// debug log
LogLvl(Lvl:=E_LogSeverity.Debug, F_Concat4('printStart: at XS:', TO_STRING(_nPosXS), ' ', _pNewAttached^.print(0)));  // print container
LogLvl(Lvl:=E_LogSeverity.Debug, F_Concat4(
                                      F_Concat3('> XS = X0(', TO_STRING(iCT.GetPosX0(iTracker:=_iCTTracker)), ')'),
                                      '',
                                      F_Concat3(' + shStartOffs(', TO_STRING(F_MeterToSubPixel(fPrintStartOffset, _fPrintResolution*_fSubPxResolution)), ')'),
                                      F_Concat3(' - shDropComp(', TO_STRING(F_MeterToSubPixel(fbDropSpeedComp.fDropPlacementError, _fPrintResolution*_fSubPxResolution)), ')')
                                   ));

// debug history
FOR i:=0 TO nC_HistorySize-1 DO sRepeatHistory[i].bSelected := FALSE; END_FOR   // clear selection
nRepeatCt := (nRepeatCt + 1) MOD nC_HistorySize;
sRepeatHistory[nRepeatCt].bSelected      := TRUE;
sRepeatHistory[nRepeatCt].nX0            := _nPosXS;
sRepeatHistory[nRepeatCt].fLen           := _pNewAttached^.pJob^.fImageDepth;  // + PrePost?
sRepeatHistory[nRepeatCt].fLenEffective  := _nPosXS - sRepeatHistory[SEL(nRepeatCt=0, nRepeatCt-1, nC_HistorySize-1)].nX0;
END_METHOD

PROPERTY bGridWasLimited : BOOL
GET
bGridWasLimited := _bGridWasLimited;
END_GET
END_PROPERTY

PROPERTY bJobActive : BOOL
GET
bJobActive := _bJobActive;
END_GET
END_PROPERTY

PROPERTY bPausePrintCanEx : BOOL
GET
bPausePrintCanEx := FALSE; //Not implemented
END_GET
END_PROPERTY

PROPERTY bPcEnabled : BOOL
GET
bPcEnabled := fB_PcAdapter.bPcEnable;
END_GET
END_PROPERTY

PROPERTY bPrintEnabled : BOOL
GET
bPrintEnabled := _bEnable;
END_GET
END_PROPERTY

PROPERTY bPrinting : BOOL
GET
bPrinting := fbPa.bPrinting;
END_GET
END_PROPERTY

PROPERTY bPrintReady : BOOL
GET
bPrintReady := fbPa.bReady;
END_GET
END_PROPERTY

PROPERTY bQueueEmpty : BOOL
GET
bQueueEmpty := NOT fB_PcAdapter.bJobValid;
END_GET
END_PROPERTY

PROPERTY bStartPrintCanEx : BOOL
GET
bStartPrintCanEx := fbPa.bStartCanEx;
END_GET
END_PROPERTY

PROPERTY bStopPrintCanEx : BOOL
GET
bStopPrintCanEx := fbPa.bStopCanEx;
END_GET
END_PROPERTY

{attribute 'monitoring':='call'}
PROPERTY bWorkerEnable : BOOL
GET
bWorkerEnable := SUPER^.bWorkerEnable;
END_GET
SET
IF _pAdsPg = 0 THEN
  SUPER^.bWorkerEnable := bWorkerEnable;
ELSE
  // mask worker enable with group enable
  SUPER^.bWorkerEnable := bWorkerEnable AND _pAdsPg^.bEnable;  
END_IF
END_SET
END_PROPERTY

{attribute 'monitoring':='call'}
PROPERTY bWorkerPrintEnable : BOOL
GET
bWorkerPrintEnable := _bWorkerPrintEnable;
END_GET
SET
_bWorkerPrintEnable := bWorkerPrintEnable;
END_SET
END_PROPERTY

(*
  Check timing for grid stream. 
  Reports an error if grid stream is too slow (machine running too fast for streaming the grid points over PDI)
  :returns: TRUE on error
*)
METHOD PRIVATE checkGridTiming : BOOL
VAR_INPUT
  nPosXS : DINT;
  nPosNow : DINT;
END_VAR
// check for timing problems
IF fMasterSpeed <> 0 THEN

  // - check pre-charge at beginning
  IF _fColumnsToPrecharge * fC_GRIDPOINT_STREAM_TIME * _sPhGridHwCfg.nGridRoiRows >= F_SubPixelToMeter(lPosSubPx:=SEL(nPosXS-nPosNow>0, 0, nPosXS-nPosNow), fResSubPx:=_fPrintResolution*_fSubPxResolution) / fMasterSpeed  THEN
    checkGridTiming := TRUE;
    LogError('Machine too fast for grid stream (for pre-charge at attach)');
  END_IF
  
  // - check charge time needed per columns vs machine speed and grid-sizeY
  IF fC_GRIDPOINT_STREAM_TIME * _sPhGridHwCfg.nGridRoiRows >= F_SubPixelToMeter(lPosSubPx:=TO_DINT(sDefGridSettings.nGridPitchX), fResSubPx:=_fPrintResolution) / fMasterSpeed THEN
    checkGridTiming := TRUE;
    LogError('Machine too fast for grid stream (time rows per column)');
  END_IF

END_IF
END_METHOD

(*
  Check if intended print position is valid. 
  - Reports an error if print start position is not in the future
  :returns: TRUE on error
*)
METHOD checkPrintposTiming : BOOL
VAR_INPUT
  nStartPos   : DINT;   // intended start position
  nCurrentPos : DINT;   // current position
END_VAR
IF (nStartPos - nCurrentPos) < 0 THEN 
  checkPrintposTiming := TRUE;
  LogWarning(Msg:=F_Concat4('Print start position:', TO_STRING(nStartPos) ,' < Encoder position:', TO_STRING(nCurrentPos)));
END_IF
END_METHOD

// apply other corrections to camera correction/deformation
METHOD PRIVATE correctionApply : BOOL
VAR_INPUT
  pPoint : POINTER TO ST_DeformationPointAccurate;
END_VAR
VAR
  i : UDINT;
END_VAR

// here apply all PU specific corrections
// - mechanical stretch based on temperature extension (if not done in Camera)
// - banana correction
// - Y-shifts of PU
// - trapzedoial correction
// - ...


// PU Deformation correction
IF GVL_Deformation.bC_UsePUDeformation THEN
  FOR i:=1 TO nPointCorrections DO
    iPointCorrections[i].updateCorrection(pPoint:=pPoint);
  END_FOR
END_IF
END_METHOD

(*
  Limit correction to boundaries
  :return: TRUE if limited
*)
METHOD PRIVATE correctionLimit : BOOL
VAR_INPUT
  pPoint : POINTER TO ST_DeformationPointAccurate;
  pCT    : POINTER TO FB_ContainerDefGrid;
END_VAR
VAR
  bLimited : BOOL;
  nExeedX, nExeedY : LREAL;
END_VAR
// limit point correction to boundaries and inform
IF pPoint^.dx >= _fLimitCorrectionX    THEN nExeedX := pPoint^.dx; pPoint^.dx := _fLimitCorrectionX;    bLimited:=TRUE; END_IF
IF pPoint^.dx <= -1*_fLimitCorrectionX THEN nExeedX := pPoint^.dx; pPoint^.dx := -1*_fLimitCorrectionX; bLimited:=TRUE; END_IF
IF pPoint^.dy >= _fLimitCorrectionY    THEN nExeedY := pPoint^.dy; pPoint^.dy := _fLimitCorrectionY;    bLimited:=TRUE; END_IF
IF pPoint^.dy <= -1*_fLimitCorrectionY THEN nExeedY := pPoint^.dy; pPoint^.dy := -1*_fLimitCorrectionY; bLimited:=TRUE; END_IF

IF bLimited THEN
  LogLvl(Lvl:=E_LogSeverity.Debug, Msg:=F_Concat4( F_concat2('Correction limited - Point=',TO_STRING(pPoint^.index)),
                                                     F_Concat5(' (c:',TO_STRING(pPoint^.col),'/r:',TO_STRING(pPoint^.row), ') '),
                                                     F_Concat4('dx:', TO_STRING(nExeedX), 'px dy:', TO_STRING(nExeedY)),
                                                     F_Concat4('px dx_max=+/-', TO_STRING(_fLimitCorrectionX), ' dy_max=+/-', TO_STRING(_fLimitCorrectionY))
                                                  ));
END_IF

_bGridWasLimited := SEL(bLimited, FALSE, TRUE);
correctionLimit := bLimited;
END_METHOD

// current job image length in [m]
PROPERTY fImageLength : LREAL
GET
fImageLength := _fCurrentImgDepth;
END_GET
END_PROPERTY

PROPERTY fMaxPrintSpeed : LREAL
GET
fMaxPrintSpeed := 0;  // TODO: when i_pc_adapter has the info from pc/ph
END_GET
END_PROPERTY

(*
  Max. supported speed [m/s], 0 if not available
*)
{attribute 'monitoring':='call'}
PROPERTY fMaxSpeed : LREAL
GET
VAR
  nSpeedMpMin : DINT;
END_VAR
nSpeedMpMin := SEL(bWorkerEnable AND _pAdsPg <> 0, 0, _pAdsPg^.lMaxPrintSpeed);
fMaxSpeed := TO_LREAL(nSpeedMpMin)/60;
END_GET
END_PROPERTY

{attribute 'monitoring':='call'}
PROPERTY fStartShiftFactor : LREAL
GET
fStartShiftFactor := _fStartShiftFactor;
END_GET
SET
_fStartShiftFactor := fStartShiftFactor;
END_SET
END_PROPERTY

{attribute 'monitoring':='call'}
PROPERTY fStartShiftOffset : LREAL
GET
fStartShiftOffset := _fStartShiftOffset;
END_GET
SET
_fStartShiftOffset := fStartShiftOffset;
END_SET
END_PROPERTY

METHOD PROTECTED gridUpdate : BOOL
VAR_INPUT
  bEnableDeformation : BOOL;      // enable correction update, else correction (0/0) is written
  pCT : POINTER TO FB_ContainerDefGrid;
  pCTHdlData : POINTER TO ST_WorkerDefGrid_CTData;
  pMaxDx : POINTER TO LREAL;
END_VAR
VAR
  bOK : BOOL;
  fCurrentColumnPos  : LREAL; // Currently column position (of current ct)
END_VAR


//TODO: rewrite this method to look cleaner (less if else)
IF sDefGridSettings.nGridSizeX  = 0 THEN RETURN; END_IF          // avoid endless loops
IF sDefGridSettings.nGridSizeY  = 0 THEN RETURN; END_IF
IF sDefGridSettings.nGridPitchX = 0 THEN RETURN; END_IF
IF pCT = 0 THEN RETURN; END_IF
IF pCTHdlData = 0 THEN RETURN; END_IF

gridUpdate:=TRUE;

// calculate grid column position
fCurrentColumnPos := pCTHdlData^.fPosRelToAttach / (sDefGridSettings.nGridPitchX * _fSubPxResolution);   // calc grid column position relative to worker

// Check for next correction update
bOK := TRUE;
IF pCTHdlData^.nChargedCols <= sDefGridSettings.nGridSizeX THEN
  IF bEnableDeformation THEN 
    // sync deformation points
    bOK := streamCorrection(pCT:=pCT,
                            fColPos := fCurrentColumnPos, 
                            pChargedCols:=ADR(pCTHdlData^.nChargedCols), 
                            pMaxDx:=pMaxDx,
                            nAvailPoints:=pCT^.nAvailableGridPoints);
  ELSE
    // sync empty deformation points (with NO correction)
    bOK := streamNoCorrection(pChargedCols:=ADR(pCTHdlData^.nChargedCols));
  END_IF
  
END_IF

gridUpdate := bOK;
END_METHOD

METHOD InitWorkerPrint : BOOL
VAR_INPUT
  pAdsPg                : POINTER TO FB_ADS_PG;       // pg ads reference (worker prints ads)
  iDefGridParamMediator : I_ParamMediator;            // for deformation settings
  fLimitCorrectionX     : LREAL;                      // correction limit in y (abs) [px]
  fLimitCorrectionY     : LREAL;                      // correction limit in y (abs) [px]
END_VAR
IF NOT bInitialized            THEN LogError('Base Worker not initialized! call init() before'); RETURN; END_IF
IF pAdspg = 0 THEN LogError('InitWorkerPrint: invalid parameter proviced'); RETURN; END_IF
IF iDefGridParamMediator = 0   THEN bInitialized := FALSE; LogError('Invalid parameter, no valid param mediator'); RETURN; END_IF

// Worker specific init
_pAdsPg := pAdsPg;
_iParamMediator := iDefGridParamMediator;

_fLimitCorrectionX := ABS(fLimitCorrectionX);
_fLimitCorrectionY := ABS(fLimitCorrectionY);

// Print Aggregate
fbPa.bSyncAfterDone := FALSE;
fbPa.init(iPcAdapter := fB_PcAdapter, iPsInterface := fbPs);
END_METHOD

METHOD mJobPause
END_METHOD

METHOD   mJobStart
VAR_INPUT
	sJobDef	: CalmarCompPrint.I_JobDefinition;
END_VAR
// Config workers static variables
// - security release position (2 * Image Length)
_fCtSecurityReleasePos := F_MeterToSubPixel(fPosMeter:=2.1*(sJobDef.fImageDepth/1000), fResoSubPx:=_fPrintResolution*_fSubPxResolution);

IF NOT bWorkerEnable THEN RETURN; END_IF  // only if enabled

// an initial definition at jobStart/(activation)
fbPs.setupObject(nObjId:=1, nCopy:=1, bStop:=FALSE, bDir:=FALSE, nPrintStartPos:=0, nImageSelection:=0, nShiftedStartX:=0);
fbPa.jobStart(bEndless:=sJobDef.isEndless());

_fCurrentImgDepth := sJobDef.fImageDepth/1000;
_bEndless := sJobDef.isEndless();
bBuffStopBit := NOT _bEndless;

// update deformation limit by job setting
//_fLimitCorrectionX   // [px]

// grid settings update
IF _iPhGrid <> 0 THEN _sPhGridHwCfg := _iPhGrid.getGridHwCfg(); END_IF 

_bJobActive := TRUE;
END_METHOD

METHOD  mJobStop
VAR_INPUT
	sStatus	: CalmarCompPrint.I_JobStatus;
END_VAR
fbPa.jobStop();
_bJobActive := FALSE;
_bPaStarted := FALSE;
_bPaStartRequested := FALSE;
END_METHOD

METHOD mProduced
VAR_INPUT
	(* current progress*)
	sProgress	: CalmarCompPrint.I_JobProgress;
END_VAR
END_METHOD

// register additional grid correction handlers
METHOD RegisterGridCorrection : BOOL
VAR_INPUT
  iGridCorrection : I_GridPointCorrection;
END_VAR
VAR
  i : UDINT;
END_VAR
IF iGridCorrection = 0 THEN LogError('registerGridCorrection: ivalid interface, ignore'); RETURN; END_IF
IF nPointCorrections >= nC_NUM_POINTCORRECTIONS THEN LogError('registerGridCorrection: too many corrections registred, ignore'); RETURN; END_IF

nPointCorrections := nPointCorrections + 1;
iPointCorrections[nPointCorrections] := iGridCorrection;
END_METHOD

METHOD registerPc : BOOL
VAR_INPUT
  iNewPC : I_PC;
END_VAR
registerPc := fB_PcAdapter.registerPc(iNewPC := iNewPC);
END_METHOD

METHOD registerPh : BOOL
VAR_INPUT
  iPH : I_PH;
END_VAR
//Attach head to print station
IF iPH <> 0 THEN
  fbPs.registerPh(iNewPh:=iPH);
  _iPhGrid := iPH.iGridCorrection;
END_IF
END_METHOD

(*
  Release CT from Worker.
  :return: TRUE if CT was released, FALSE if no CT was registered 
*)
METHOD Release : BOOL
VAR_INPUT
  iCT              : I_CT;                         (*container at triggered event position*)
END_VAR

Release := SUPER^.Release(iCT:=iCT);
END_METHOD

// Release all attached CTs
METHOD PRIVATE ReleaseAllAttached
VAR
  i : UDINT;
  pCt : POINTER TO FB_ContainerDefGrid;
END_VAR
//Work only with attached container
IF _nAttachedCTs = 0 THEN RETURN; END_IF
  
FOR i:=nLowerIndexCTList TO nLowerIndexCTList + _nAttachedCTs - 1 DO
  pCt := _pAttachedCTList[i];
  pCt^.AbortDeformation(sReason:=EC_Print.ecPaAbortHold.Desc, Src:=_pEcSrc^, bHideLog:=TRUE);
  
  Release(iCT:=pCt^);
END_FOR
END_METHOD

METHOD PRIVATE setupPosition
VAR
  fPreStartShift : LREAL;
  fCalculatedWorkerPos : LREAL;
END_VAR
IF _pAttachedCt <> 0 THEN RETURN; END_IF   // Update only without attached container

// Worker position update
fPreStartShift := (_fStartShiftOffset + _fStartShiftFactor * fMasterSpeed);
fCalculatedWorkerPos := fPrintStartOffset + fPreStartShift;
IF _fWorkerPosition <> fCalculatedWorkerPos THEN   // Worker position changed
  fPosition := fCalculatedWorkerPos;  // Update worker position
END_IF
END_METHOD

METHOD PRIVATE sim
END_METHOD

METHOD PRIVATE streamCorrection : BOOL
VAR_INPUT
  pCT : POINTER TO FB_ContainerDefGrid;
  fColPos : LREAL;  // current column position (relative to Attach-Pos)
  pChargedCols : POINTER TO UDINT;  // number of already charged columns (pointer for internal edit)
  pMaxDx : POINTER TO LREAL;
  nAvailPoints : UDINT;     // available gridPoints on CT
END_VAR
VAR
  nRow : UDINT;
  bWasSet : BOOL;
  sPoint : ST_DeformationPointAccurate;
  fCurrentPreCharge  : LREAL; // Currently to be precharged (for scope)
END_VAR
VAR_INST
  nAvailPoints_mem : UDINT;
END_VAR
IF pChargedCols = 0 THEN RETURN; END_IF

streamCorrection := TRUE;

fCurrentPreCharge := fColPos + _fColumnsToPrecharge;

WHILE pChargedCols^ < LIMIT(0, FLOOR(fCurrentPreCharge), sDefGridSettings.nGridSizeX) DO
  
  IF nAvailPoints >= sDefGridSettings.nGridSizeY * (pChargedCols^+1) THEN     // Complete next column available?
    
    nAvailPoints_mem := 0;
    LogLvl(Lvl:=E_LogSeverity.Debug, Msg:=F_Concat4('CT: ', TO_STRING(pCT^.pCT^.iId),' Charge CG col: ', TO_STRING(pChargedCols^)));
    
    pMaxDx^ := 0;   // per columns
    
    FOR nRow := 0 TO sDefGridSettings.nGridSizeY - 1 DO
      
      // get points
      IF pCT^.getDeformationPoint(nCol:=pChargedCols^, nRow:=nRow, nSel:=0, sPoint=>sPoint, bWasSet=>bWasSet) THEN
        
        IF NOT bWasSet THEN LogWarning(F_Concat5('Point[c(',TO_STRING(pChargedCols^),')/r(', TO_STRING(nRow),')] was not set')); END_IF
        
        // apply PU corrections
        correctionApply(pPoint:=ADR(sPoint));
        
        // limitation corrections
        correctionLimit(pPoint:=ADR(sPoint), pCT:=pCt);
        
        // max. dx tracing
        IF sPoint.dx > pMaxDx^ THEN pMaxDx^ := sPoint.dx; END_IF
        
        // send point
        IF NOT fbPs.newGridPoint(sPoint:=sPoint) THEN
          // err
          LogError(Msg:='stream new point failed');
          streamCorrection:=FALSE;
          RETURN;
        ELSE
          // ok
          pCT^.storeStreamedDeformationPoint(pPoint:=ADR(sPoint));    // save to sent table
          IF bEnVerbose THEN
            F_Concat3( 
              F_concat2('Send Point=',TO_STRING(sPoint.index)),
              F_Concat5(' (c:',TO_STRING(sPoint.col),'/r:',TO_STRING(sPoint.row), ')'),
              F_Concat4(' dx=', TO_STRING(sPoint.dx), ' dy=', TO_STRING(sPoint.dy))
            );
          END_IF
        END_IF
      ELSE
        LogError(Msg:='get new grid point failed');
        streamCorrection:=FALSE;
      END_IF
    END_FOR
    
    pChargedCols^ := pChargedCols^ + 1;
  ELSE
    
    // not yet enought points for next full column
    IF nAvailPoints > nAvailPoints_mem THEN // log once or after every update of new available points
      LogLvl(Lvl:=E_LogSeverity.Error, Msg:=F_Concat3(
                                            F_Concat2('CT: ', TO_STRING(pCT^.pCT^.iId)), 
                                            F_Concat2(' Print column expected but not available. Avil=', TO_STRING(nAvailPoints)),
                                            F_Concat2(' of expected: ', TO_STRING(sDefGridSettings.nGridSizeY * (pChargedCols^+1)))
                                          ));
    END_IF
    nAvailPoints_mem := nAvailPoints;
    streamCorrection:=FALSE;
    RETURN;
  END_IF
  
END_WHILE
END_METHOD

METHOD PRIVATE streamNoCorrection : BOOL
VAR_INPUT
  pChargedCols : POINTER TO UDINT;  // number of already charged columns (pointer for internal edit)
END_VAR
VAR
  nRow : UDINT;
  sPoint : ST_DeformationPointAccurate;
END_VAR
IF pChargedCols = 0 THEN RETURN; END_IF

// send points with no deformation
FOR nRow := 0 TO sDefGridSettings.nGridSizeY - 1 DO
    MEMSET(destAddr:=ADR(sPoint), fillByte:=0, n:=SIZEOF(sPoint));
    sPoint.col := TO_DINT(pChargedCols^);
    sPoint.row := TO_DINT(nRow);
    IF NOT fbPs.newGridPoint(sPoint:=sPoint) THEN
       LogError(Msg:='stream new point failed');
       streamNoCorrection:=FALSE;
       RETURN;
    END_IF
END_FOR

// select next column
pChargedCols^ := pChargedCols^ + 1;

streamNoCorrection := TRUE;
END_METHOD

METHOD work
VAR
  bDeformErr : BOOL;
  nDeformStep : E_DeformationStep;
  i : UDINT;
  pCt : POINTER TO FB_ContainerDefGrid;
  pCtHdlData : POINTER TO ST_WorkerDefGrid_CTData;
  nUpdateStopPos : DINT;
  fMaxDx : LREAL;
END_VAR
IF _iParamMediator = 0 THEN F_Report_Error(ErrType:=EN_REPORT_ERROR_TYPE.Report_Error_0Pointer); RETURN; END_IF
bError := FALSE; nError := 0;

setupPosition();  // calculate and set worker position

SUPER^.work();

(*Print correction*)
fbDropSpeedComp(fMasterSpeed:=fMasterSpeed, fDropTravelDistance:=fPUElevation);

(*Update virtual encoder on all controller boards*)
fB_PcAdapter.setEncoderPos(nPrintPos);
fB_PcAdapter();

(*Call print aggregate*)
rTrigHwSync(CLK:=bHardwareSync); 
IF rTrigHwSync.Q THEN fbPa.sync(); END_IF   // external sync cmd

// PA control
fbPa.bHold := bHardwareHold;                // external hw hold, NOTE: this stop the current print iPC.stop()
fbPa();
PaStartTimeout(IN:=_bPaStartRequested, PT:=fbPa.fbStatePrepare.tC_PrepareTimeout+T#10MS);

IF _bPaStartRequested THEN
  // Starting...
  IF fbPa.bPrinting THEN
    // started
    _bPaStarted := TRUE; 
    _bPaStartRequested := FALSE;
  ELSIF PaStartTimeout.Q THEN     // Abort print
    // start timeout -> abort
    _bPaStarted := FALSE;
    _bPaStartRequested := FALSE;
    fbPa.printStop(bSyncedStop:=FALSE);
    ReleaseAllAttached();
  END_IF
ELSIF _bPaStarted THEN
  // - Started... Supervision of FSM
  IF fbPa.bDone OR fbPa.bStop THEN  // if pa did stop
    _bPaStarted := FALSE; 
    ReleaseAllAttached();
  (*ELSIF fbpa.bError THEN
    ReleaseAllAttached();*)
	END_IF 
  // - disabled
  IF NOT bWorkerEnable THEN
    _bPaStarted := FALSE;
    fbPa.printStop(bSyncedStop:=FALSE);
    ReleaseAllAttached();
  END_IF
  // - machine stopped
  IF bFastStopRequest OR bHardwareHold THEN
    _bPaStarted := FALSE;
    fbPa.printStop(bSyncedStop:=FALSE);
    ReleaseAllAttached();
	END_IF
  // - Synced stopping request
  IF bPrintStopRequest THEN
    IF NOT _bPaStopping THEN  _bPaStopping := TRUE;
      fbPs.stopObject(nObjId:=0, 
                      nStopPosition:=   _nPosXS           // use last used/calculated XS
                                      + F_MeterToSubPixel(fPosMeter:=_fCurrentImgDepth + 0.05, fResoSubPx:=_fPrintResolution*_fSubPxResolution)
                                      + TO_DINT(nPhDepth*_fSubPxResolution));
      fbPa.printStop(bSyncedStop:=TRUE);                  // should stop automatically when all buffer are done   
     END_IF
  ELSE
    _bPaStopping := FALSE;
  END_IF
END_IF

bPrintActive := _bPaStarted;


// for all attached CTs ----------------
// - Disable      -> PA.Stop, tag all as error, release all [OK]
// - FastStop     -> PA.Stop, tag all as error, release all [  ]
// - Hold         -> PA.Hold => PC.stop() [  ]
// - PA Starting  ->  [  ]
// - JobStop      -> PA.jobStop() -> tag all as error, release all [  ]
// - Normal Stop  -> PS.Request a stop [  ]
// - OK           =>  GridStream -> Release when all done [  ]
FOR i:=nLowerIndexCTList TO nLowerIndexCTList + _nAttachedCTs - 1 DO
  pCt := _pAttachedCTList[i];
  // Handling Data
  // - fPosRelToAttach: position relative to attach
  // - nChargedCols: charged columns
  // - nData2: not used
  // - fData1: not used
  // - fData2: not used
  pCtHdlData := ADR(_stAttachedCTData[i]);
  
  // Grid update
  bDeformErr := pCt^.getDeformationStatus(eDStep=>nDeformStep);
  IF NOT bDeformErr AND nDeformStep >= E_DeformationStep.gridStarted AND NOT _bForceDefGridOff THEN
    IF NOT gridUpdate(bEnableDeformation:=TRUE, pCT:=pCt, pCTHdlData:=pCtHdlData, pMaxDx:=ADR(fMaxDx)) THEN
      pCt^.AbortDeformation(sReason:='deformation point update failed', Src:=_pEcSrc^, bHideLog:=FALSE);
    END_IF
  ELSE
    // not started or error already --> erase deformation points and send no correction points
    IF NOT gridUpdate(bEnableDeformation:=FALSE, pCT:=pCt, pCTHdlData:=pCtHdlData, pMaxDx:=ADR(fMaxDx)) THEN
      pCt^.AbortDeformation(sReason:='deformation point update failed', Src:=_pEcSrc^, bHideLog:=FALSE);
    END_IF
  END_IF
  
  // RELEASE when Grid stream finished
  IF pCtHdlData^.nChargedCols >= sDefGridSettings.nGridSizeX THEN
    IF NOT _bEndless THEN // single print mode
      // Update print length in single print mode
      nUpdateStopPos := pCtHdlData^.nXS                                                                                   // XS print start position
                      + F_MeterToSubPixel(fPosMeter:=_fCurrentImgDepth, fResoSubPx:=_fPrintResolution*_fSubPxResolution)  // sheet length
                      + F_MeterToSubPixel(fPosMeter:=fMaxDx, fResoSubPx:=_fPrintResolution)                               // max. deformation
                      + TO_DINT(nPhDepth*_fSubPxResolution);
      fbPs.stopObject(nObjId:=0, nStopPosition:=nUpdateStopPos);        // update (overwrite firmware internal calculated) jm stop position
      LogLvl(Lvl:=E_LogSeverity.Debug, Msg:=F_Concat6('Update StopPos=', TO_STRING(nUpdateStopPos),' (',F_UDINT_TO_HEXSTR(lVal:=TO_UDINT(nUpdateStopPos), bLower:=FALSE), ') on ', pCt^.print(format:=0)));
    END_IF
    Release(pCt^);
  END_IF
END_FOR


// forward pa state to pg ads
IF _pAdsPg <> 0 THEN
  _pAdsPg^.aState := fbPa.aPaState;
  _pAdsPg^.lError := nError; 
  _pAdsPg^.bError := bError;
END_IF


// logging config
fbPa.LogLevel := LogLevel;
fB_PcAdapter.LogLevel := LogLevel;

sim();
END_METHOD

END_FUNCTION_BLOCK

// ---- POUs/Print/WEU/FB_PrintModule_WEU_View.TcPOU
FUNCTION_BLOCK FB_PrintModule_WEU_View
VAR
  // helper
  bInit   : BOOL;
  
  // config
  _pModule : POINTER TO FB_PrintModule_WEU;
  _pPositioning : POINTER TO FB_PrintPositionDmax;
  
  fbCTTrackerView : FB_CTTrackerView;
  
  // view selections
  nSelWorkerPrint : UDINT := 1;
  bShowFineAlignement : BOOL;
  // hardware view
  bShowPhDetail : BOOL;
  nSelPhDetail : UDINT := 1;
  bShowPcDetail : BOOL;
  nSelPcDetail : UDINT := 1;
  
  // motion and position view
  bShowPositionDetail : BOOL;
  bMovingInd : BOOL;
  fSpeed  : LREAL;
  fbBlink_Moving : FB_BLINK;
  
  // debug view
  bShowDebugAndSim : BOOL;
  
  fbBlink_Printing : FB_BLINK;
  bBlinkPrint : BOOL;
  bPrintInd : ARRAY[1..GVL_WEU.nC_MaxWorkerPrintPerPm] OF BOOL;
  fMaxPos : LREAL;
  t : TIME;
  zPos_PM : UDINT;
  i : UDINT;
END_VAR

VAR CONSTANT
  nC_MAX_WORKER_VIEWS : UINT := 10;
END_VAR

IF NOT checkConfig() THEN RETURN; END_IF    // check config

// -- show moving -----------------------
fSpeed := _pPositioning^.getSpeed();
IF LrealIsNaN(x:=fSpeed) THEN
  fSpeed := 0;
END_IF
t := LREAL_TO_TIME(1000-fSpeed*900);
fbBlink_Moving(bI_Enable:=SEL(fSpeed > 0, FALSE, TRUE), tI_Time:=t, bO_Out=>bMovingInd);

t := T#400MS;
fbBlink_Moving(bI_Enable:=TRUE, tI_Time:=t, bO_Out=>bBlinkPrint);
FOR i:=1 TO GVL_WEU.nC_MaxWorkerPrintPerPm DO
  bPrintInd[i] := _pModule^.fbWorkerPrint[i].bPrinting AND bBlinkPrint;
  fMaxPos := MAX(_pModule^.fbWorkerPrint[i].fPosition, fMaxPos);
END_FOR


// -- show pm module position
zPos_PM := SEL(_pModule^._pModuleMachineState^.bUnitInPrintPosition, 0, 40);

// -- show pg in p,
nSelWorkerPrint := LIMIT(1, nSelWorkerPrint, GVL_WEU.nC_MaxWorkerPrintPerPm);

// -- show ph detail
nSelPhDetail := LIMIT(1, nSelPhDetail, _pModule^._nPh);
nSelPcDetail := LIMIT(1, nSelPcDetail, _pModule^._nPc);

// -- CTTracker overview view
fbCTTrackerView.fX_m  := fMaxPos + 0.1;
fbCTTrackerView.fY_m  := 1;
fbCTTrackerView.nX_px := 300;
fbCTTrackerView.nY_px := 100;
fbCTTrackerView.fPxToMRatio := fbCTTrackerView.nX_px / fbCTTrackerView.fX_m;
fbCTTrackerView.iPrintPosition :=_pPositioning^;
fbCTTrackerView();

METHOD checkConfig : BOOL
VAR_INPUT
END_VAR
VAR_INST
  _fX_m, _fY_m   : LREAL;
  _nX_px, _nY_px : DINT; 
END_VAR
VAR
  bOK : BOOL;
END_VAR
IF NOT bInit THEN RETURN; END_IF

checkConfig := TRUE;
END_METHOD

METHOD init : BOOL
VAR_INPUT
  pModule : POINTER TO FB_PrintModule_WEU;
  pPositioning : POINTER TO FB_PrintPositionDmax;
END_VAR
IF pPositioning = 0 OR pModule = 0 THEN RETURN; END_IF

_pModule := pModule;
_pPositioning := pPositioning;

// cttracker overview
fbCTTrackerView.init(pCTTracker:=ADR(_pModule^.fbCTTracker));

bInit := TRUE;
END_METHOD

END_FUNCTION_BLOCK

// ---- POUs/Print/obsolete/FB_DRIFTCONTROL.TcPOU
FUNCTION_BLOCK FB_DRIFTCONTROL
VAR_INPUT
  bI_Reset                    : BOOL;            (*reset fb and controller*)
  bI_Enable                   : BOOL;            (*[internal] auto enable of control*)
  bI_OutputEnable             : BOOL;            (*enable control output or 1.0 if off*)
  bI_RegisterMark             : BOOL;            (*start trigger (e.g. register mark)*)
  
  lI_RegisterMarkPosition     : DINT;            (*[Subpixel] Mark position*)
  lI_RefPosition              : DINT;            (*[Subpixel] Refereence position*)
  lI_ImgPosition              : DINT;            (*[Subpixel] Image position*)
(*UNUSED*)  fI_RefPosition            : LREAL;          (*[um] Refereence position*)    
(*UNUSED*)  fI_ImgPosition            : LREAL;          (*[um] Image position*)

  iI_Res_Ph                   : INT;             (*[dpi] resolution printhead native*)
  iI_Res_SubPix               : INT;             (*[-] resolution subpixel*)
  pI_JobSettings              : POINTER TO ST_JobSettings;
  
  fI_ControllerPGain          : LREAL := 0.5;    (*PDI controller P-Gain*)
  fI_ControllerIGain          : LREAL := 20;     (*PDI controller I-Gain*)
  
  fI_DriftTimeShift           : LREAL;           (*[ms] register shift time*)
  fI_TaskCycleTime            : REAL;            (*Task cycle time of actual task [s]*)
END_VAR

VAR_OUTPUT
  fO_SpeedCorrectionFactor    : LREAL;           (*[-] controller output*)
  bO_ContrErr                 : BOOL;            (*correction fail (out of bound)*)
  bO_SupervisionContrErr      : BOOL;            (*supervision (out of bound)*)
END_VAR

VAR
  bL_ControlActive            : BOOL;
  bL_RegisterMark             : BOOL;
  
  lL_LastRegisterMarkPosition : DINT;            (*[SubPixel] last stored mark position*)
  lL_LastRefPosition          : DINT;            (*[Subpixel] Refereence position*)
  lL_LastImgPosition          : DINT;            (*[Subpixel] Image position*)

  fL_RefSpeed                 : LREAL;           (*[rev/s] : rev ^= image, revolution of reference axe sync with image*)
  fL_ImgSpeed                 : LREAL;           (*[rev/s] : rev ^= image, revolution of reference axe sync with image*)
  fL_RefLength                : LREAL;           (*[Subpixel in float!] real length of one image = reference distance between print marks*)
  lL_ImgLength                : DINT;            (*[Subpixel] image length of job*)
  fL_RefPos                   : LREAL;           (*[rev] : 1rev ^= 1ImageLength, number rev after start*)
  fL_ImgPos                   : LREAL;           (*[rev] : 1rev ^= 1ImageLength, number rev after start*)
  fL_LastRefPos               : LREAL;           (*[rev] : 1rev ^= 1ImageLength, number rev after start*)
  fL_LastImgPos               : LREAL;           (*[rev] : 1rev ^= 1ImageLength, number rev after start*)
  fL_ShiftPos                 : LREAL;           (*[rev] shift position rev->img*)

  fL_DeltaCtrl                : LREAL;           (**)
  fL_CtrlGainFactor           : LREAL;           (**)
        
  fL_DeltaTimeStamp           : LREAL;           (**)
  tL_CurrentTimeStamp         : T_DCTIME64;      (* Get Current Timestamp *)
  tL_LastTimeStamp            : T_DCTIME64;      (* Get Current Timestamp *)
  fB_PID                      : FB_BasicPID;     (**)
  iL_State                    : UINT;            (**)

  bL_FormatWarning            : BOOL;
  bL_Error                    : BOOL;
  bL_RegisterEvent            : BOOL;
  bL_ResetInternal            : BOOL;            (*internal reset*)
  fL_DeltaLength              : LREAL;           (*image length difference between img and ref bewtween a cycle*)
  lL_ConversionErrorCtr       : UDINT;

  bL_SupervisionContrErr      : BOOL;            (*supervision (out of bound)*)
  fb_TonSupervisionContrErr   : TON;             (*supervision (out of bound)*)

  fC_MaxCorrection            : LREAL := 1.10;  (*moved from Constant: org value: 1.05*)
  fC_MinCorrection            : LREAL := 0.90;  (*moved from Constant: org value: 0.95*)
  fC_MaxControlError          : LREAL := 0.2;   (*moved from Constant: org value: 0.1*)
END_VAR

VAR CONSTANT
  fC_NormSpeedCorrectionFactor: LREAL := 1.0;
  
  fC_MaxFormatDifference      : LREAL := 1.0;
  
  fC_MaxFormatLength          : LREAL := 1.0;       (*m*)
  fC_MinSubstrateSpeed        : LREAL := 5.0/60.0 ; (*m/s*)
  lC_MaxFormatLength          : DINT  := LREAL_TO_DINT(fC_MaxFormatLength/0.0254*32*600);  (*Subpixel*)
  fC_MaxCycleTime             : LREAL := fC_MaxFormatLength/fC_MinSubstrateSpeed;  (*sec*)
END_VAR

VAR PERSISTENT
  fR_SpeedCorrectionWindow    : LREAL := 0.05;     (*Supervision window*)
  tR_SpeedCorrectionTime      : TIME  := T#10S;    (*Supervision time*)
END_VAR

(*--- Reset*)
IF bI_Reset OR bL_ResetInternal THEN
  iL_State := 0;
END_IF;

(*--- cyclic called on register event*)
IF bI_RegisterMark AND NOT bL_RegisterMark THEN
  bL_RegisterEvent    := TRUE;
  tL_CurrentTimeStamp := F_GetCurDcTaskTime64();
  fL_DeltaTimeStamp   := (ULINT_TO_LREAL(tL_CurrentTimeStamp) - ULINT_TO_LREAL(tL_LastTimeStamp)) * 0.000_000_001;
ELSE
  bL_RegisterEvent    := FALSE;
END_IF


// ----- State machine 
CASE iL_State OF
  000:  (*Reset --------------------*)
    bL_ControlActive:=FALSE;
    fB_PID(bReset := TRUE);
    fO_SpeedCorrectionFactor:=1.0; 
    fB_PID.bReset:=FALSE;
    fL_RefPos:=0;
    fL_ImgPos:=0;

    IF pI_JobSettings<>0 THEN
      iL_State:=001;
    ELSE
      iL_State:=000;
    END_IF

    bL_ControlActive:=0;
    bL_Error:=FALSE;
     bI_Enable:=FALSE; (*Disable by default*)
    bO_ContrErr := FALSE;
    
  001:  (*Control Disabled --------------------*)
    (*New PrintLib 1.5.2.6
    lL_ImgLength:=UDINT_TO_DINT(pI_JobSettings^.lI_ImageDepth)*iI_Res_SubPix; *)
    lL_ImgLength := FC_CONV_M_TO_SUBPX( UDINT_TO_LREAL(pI_JobSettings^.lI_ImageDepth) / 1_000_000
                                      , iI_Res_Ph
                                      , iI_Res_SubPix
                                      , ADR(PRG_SYSTEMBASE.lI_ConversionErr));

    IF pI_JobSettings^.lI_PrintMode.ePr_PRINT_MODE_ENDLESS THEN
      bI_Enable:=TRUE; (*Automatically enable in Endless Mode*)
    END_IF    
    
    IF bI_Enable AND (fL_DeltaTimeStamp < fC_MaxCycleTime) AND bL_RegisterEvent AND lL_ImgLength >0 THEN (*Enabled and moving*)
      iL_State:=010;
    ELSE
      iL_State:=001;
    END_IF
    fO_SpeedCorrectionFactor:=1.0; 

  010:  (*Starting Controller ------------------*)
    IF (fL_DeltaTimeStamp > fC_MaxCycleTime) THEN
      iL_State:=001;
    ELSIF bL_RegisterEvent THEN
        (*registered first label*)
      fL_RefLength := DINT_TO_LREAL(lI_RegisterMarkPosition - lL_LastRegisterMarkPosition);
      (*New PrintLib 1.5.2.6
      lL_ImgLength:=UDINT_TO_DINT(pI_JobSettings^.lI_ImageDepth)*iI_Res_SubPix; *)
      lL_ImgLength := FC_CONV_M_TO_SUBPX( UDINT_TO_LREAL(pI_JobSettings^.lI_ImageDepth) / 1_000_000
                                        , iI_Res_Ph
                                        , iI_Res_SubPix
                                        , ADR(PRG_SYSTEMBASE.lI_ConversionErr));
      
      IF fL_RefLength > 0 AND lL_ImgLength > 0 THEN
        IF DINT_TO_LREAL(ABS(FC_LREAL_TO_DINT(fL_RefLength, ADR(lL_ConversionErrorCtr))-lL_ImgLength)*100)/fL_RefLength > fC_MaxFormatDifference THEN
          bL_FormatWarning:=TRUE;
        ELSE
            bL_FormatWarning:=FALSE;
        END_IF
        iL_State:=020;
        fL_RefPos:=0;
        fL_ImgPos:=0;
      ELSE
        iL_State:=099;
      END_IF
    ELSE
      iL_State:=010;
    END_IF
    
    fL_CtrlGainFactor:=1.0;
    bL_ControlActive:=FALSE;
    
  020:  (*Controller enabled--------------------*)
    
    IF bL_RegisterEvent THEN (*run controller when a mark trigger was detected*)
      (*position in [rev] from beginning*)
      fL_RefLength := DINT_TO_LREAL(lI_RegisterMarkPosition - lL_LastRegisterMarkPosition);
      IF fL_RefLength > 0 THEN
        fL_RefPos := fL_LastRefPos + DINT_TO_LREAL(lI_RefPosition - lL_LastRefPosition) / fL_RefLength;
        fL_ImgPos := fL_LastImgPos + DINT_TO_LREAL(lI_ImgPosition - lL_LastImgPosition) / DINT_TO_LREAL(lL_ImgLength);  
      END_IF

      (*calculate current speed of ref and img position*)
      (*    'traveled pos in cycle' / ('Reference Length sampled' / 'time diff sampled' *)
      fL_RefSpeed := (fL_RefPos - fL_LastRefPos) / fL_DeltaTimeStamp;
      fL_ImgSpeed := (fL_ImgPos - fL_LastImgPos) / fL_DeltaTimeStamp;   
    
//      fL_RefSpeed:=DINT_TO_LREAL(lI_RefPosition-lL_LastRefPosition)/(fL_RefLength*fL_DeltaTimeStamp);
//      fL_ImgSpeed:=DINT_TO_LREAL(lI_ImgPosition-lL_LastImgPosition)/(DINT_TO_LREAL(lL_ImgLength)*fL_DeltaTimeStamp);    
//      fL_RefPos:=0.000001*fI_RefPosition/( fL_RefLength / INT_TO_REAL(iI_Res_Ph * iI_Res_SubPix) * 0.0254);
//      fL_ImgPos:=0.000001*fI_ImgPosition/FC_CONV_SUBPX_TO_M(lL_ImgLength,INT_TO_UDINT(iI_Res_Ph),INT_TO_UDINT(iI_Res_SubPix));
      
      (*shift calculation*)
      fL_ShiftPos := (fI_DriftTimeShift / 1000) * fL_RefSpeed;
      
      (*calc control diff*)
      fL_DeltaCtrl := (fL_RefPos - fL_ImgPos) + fL_ShiftPos;
      
      (*controller*)
      fB_PID.fCtrlCycleTime  := fL_DeltaTimeStamp;  // use fI_TaskCycleTime if running controller cyclically
      fB_PID.bReset          := FALSE;
      fB_PID.fSetpointValue  := fL_DeltaCtrl;
      fB_PID.fActualValue    := 0.0;
      fB_PID.fKp             := fI_ControllerPGain * fL_CtrlGainFactor;
      fB_PID.fTd             := 0.0;
      fB_PID.fTn             := fI_ControllerIGain;
      fB_PID.fTv             := 0.0;

      fB_PID();
    END_IF
    
    IF bI_OutputEnable THEN
      fO_SpeedCorrectionFactor := fB_PID.fCtrlOutput + 1.0;
    ELSE
      fO_SpeedCorrectionFactor := 1.0;
    END_IF;

    IF fO_SpeedCorrectionFactor > fC_MaxCorrection THEN
      fO_SpeedCorrectionFactor := fC_MaxCorrection;
      fL_CtrlGainFactor := 0.1;  (*TODO ARW*)
      bO_ContrErr       := TRUE;
    ELSIF fO_SpeedCorrectionFactor < fC_MinCorrection THEN
      fO_SpeedCorrectionFactor := fC_MinCorrection;
      fL_CtrlGainFactor := 0.1;  (*TODO ARW*)
      bO_ContrErr       := TRUE;
    ELSE
      fO_SpeedCorrectionFactor := fO_SpeedCorrectionFactor;
      fL_CtrlGainFactor := 1;
      bO_ContrErr       := FALSE;
    END_IF
    (*Supervision*)
    IF fO_SpeedCorrectionFactor > (fC_NormSpeedCorrectionFactor + fR_SpeedCorrectionWindow) THEN
      bL_SupervisionContrErr := TRUE;
    ELSIF fO_SpeedCorrectionFactor < (fC_NormSpeedCorrectionFactor - fR_SpeedCorrectionWindow) THEN
      bL_SupervisionContrErr := TRUE;
    ELSE
      bL_SupervisionContrErr := FALSE;
    END_IF
    fb_TonSupervisionContrErr( IN := bL_SupervisionContrErr, PT := tR_SpeedCorrectionTime);
    bO_SupervisionContrErr := fb_TonSupervisionContrErr.Q;
    
    (*Check for errors  while control was on*)
    IF ((fL_DeltaTimeStamp > fC_MaxCycleTime) OR (fL_DeltaCtrl > fC_MaxControlError) OR fL_RefLength=0) AND bL_RegisterEvent THEN
      iL_State:=099;
    ELSIF NOT bI_Enable THEN
      iL_State:=030;  
    ELSE
      iL_State:=020;
    END_IF
    bL_ControlActive:=TRUE;

  030:  (*Stopping controller-------------------*)
    iL_State:=001;  
    bL_ControlActive:=FALSE;
    fO_SpeedCorrectionFactor:=1.0;
    bO_ContrErr := FALSE;
    
  099:  (*Error---------------------------------*)
    bL_Error:=TRUE;
    bL_ControlActive:=FALSE;
    fO_SpeedCorrectionFactor:=1.0; 
    bO_ContrErr := FALSE;
END_CASE

(*--- cyclic called on register event*)
IF bL_RegisterEvent OR bI_Reset THEN
  (*save old values & debug*)
  fL_DeltaLength              := lL_ImgLength - fL_RefLength;  (*debug only*)
  lL_LastRegisterMarkPosition := lI_RegisterMarkPosition; 
  lL_LastRefPosition          := lI_RefPosition;       (*used for speed only*)
  lL_LastImgPosition          := lI_ImgPosition;       (*used for speed only*)
  tL_LastTimeStamp            := tL_CurrentTimeStamp;
  fL_LastRefPos               := fL_RefPos;
  fL_LastImgPos               := fL_ImgPos;
END_IF;

END_FUNCTION_BLOCK

// ---- POUs/Print/obsolete/FB_START_POS_DETECT_WEU.TcPOU
FUNCTION_BLOCK FB_START_POS_DETECT_WEU
(*************************************************************************************************)
(*  FILENAME:    FB_START_POS_DETECT_WEU                                                         *)
(*  PROJECT:     CALMAR PUPLC                                                                    *)
(*  COPYRIGHT:   All rights reserved (c) Wifag//Polytype, Fribourg/Switzerland (2016)            *)
(*  ENVIRONMENT: TwinCAT PLC                                                                     *)
(*  VERSION:     <version>                                                                       *)
(*************************************************************************************************)
(*  DESCRIPTION:                                                                   <description> *)
(*    With 1 timestamped sensors, this function that can be used with marked web,                *)
(*    will return the lateral offset of the web.                                                 *)
(*                                                                                </description> *)
(*************************************************************************************************)

VAR_INPUT
  pI_ConversionErr                : POINTER TO UDINT;  (*counts catched data type conversion overflows*)

  (*EL1252*)
  bIKp_CmdStartPrintSta     AT%I* : BOOL;        (*Command to start print station*)
  tIKp_TimeStampPos         AT%I* : T_DCTIME64;  (*TimeStamp Pos_Edge @EL1252*)
  tIKn_TimeStampNeg         AT%I* : T_DCTIME64;  (*TimeStamp Neg_Edge @EL1252*)

  (*signals*)
  bI_Sensor1_State                : BOOL;            (*Sensor 1 signal*)
  tI_Sensor1_TimeStampPos         : T_DCTIME64;      (*Sesnor 1 last detection timestamp*)
  tI_Sensor1_TimeStampNeg         : T_DCTIME64;      (*Sesnor 1 last detection timestamp*)
  iI_CurrentTimeStampComp         : DINT := 2_000;   (*µs*)
  iI_SensorTimeStampComp          : DINT := 150;     (*µs*)

  iI_CurrentPos                   : DINT;            (*current position in Pulses/Subpixels*)
  fI_ConveyorSpeed                : REAL;            (*actual speed of conveyor in [m/s]*)
  fI_SubstrateLength              : REAL;            (*length of substrate in [m]*)
  bI_Reset                        : BOOL := FALSE;   (*reset this fb*)
  bI_MissedMarks                  : BOOL := TRUE;    (*At least one sensor missed mark, detected by FB_SUPERVISOR*)
  bI_SpeedValid                   : BOOL;

  (*configuration*)
  bI_WithMark                     : BOOL := TRUE;    (*use with or without mark detection, TRUE=with detection*)
  bI_MarksInverted                : BOOL := FALSE;   (*invert in case of wrong mirrored marks*)
  fI_MarkLength                   : REAL;            (*length of detection mark [m]*)
  fI_MarkHeight                   : REAL;            (*width of detection mark [m]*)

  fI_Resolution                   : LREAL := 1;

  (*Debug & Test*)
  bI_SimTriggerActive             : BOOL;            (*Sim start trigger active*)
  bI_ManualTrigger                : BOOL;            (*Manual start trigger*)
  iI_ManualTriggerPosition        : DINT;            (*Manual trigger position [SubPx]*)
END_VAR

VAR_OUTPUT
  fO_LateralOffset                : REAL;       (*[m]*)

  iO_Offset_X0                    : DINT;       (*[SubPx]*)
  bO_StartTrig                    : BOOL;       (**)
  bO_Eject                        : BOOL;       (*Error occured, eject sheet*)
  bO_MarkDetected1                : BOOL;

  nO_PrintMarkPosBits             : WORD;       (*Print mark position (bit coded)*)
END_VAR

VAR
  (*sensor 1*)
  fL_S1_Duration                  : REAL;
  tL_S1_RisingEdge                : T_DCTIME64;
  tL_S1_FallingEdge               : T_DCTIME64;
  bL_S1_AcqOK                     : BOOL;
  fL_S1_Length                    : REAL;       (*[m]*)
  bL_memS1_State                  : BOOL;
  bL_inhibSensor1                 : BOOL;       (*inhibit sensor signals, TRUE=inhibit*)

  bL_StopCondition                : BOOL;       (*condition to send a stop trigger*)
  iL_InhibitLength                : DINT;       (*inhibit length in pulse [SubPx]*)
  fL_InhibitSubstrateDecrease     : REAL := 0.010;   (*decrease substrate for inhibit in [m]*)

  tL_CurrentTimeStamp             : T_DCTIME64; (* Get Current Timestamp *)
  fL_CurrentTimeStamp             : LREAL;
  fI_Sensor1_TimeStamp            : LREAL;

  fL_DeltaDistance                : LREAL;      (*Distance that the substrate moved between the detection and the treatment of the information [m]*)
  fL_TempVar                      : LREAL;      (*[SubPx]*)
  iL_DeltaPosition                : DINT;       (*distance [SubPx]*)
  iL_DbgDeltaP_min                : UDINT := 100_000;
  iL_DbgDeltaP_max                : UDINT := 0;

  iL_Dbg_0Div                     : UDINT := 0; (*counts all avoided zero pointer divisions*)
  iL_Dbg_MissedMarks              : DINT;

  bL_SpeedValid                   : BOOL;
  
  fb_TonCheckMarks                : TON;
END_VAR

VAR PERSISTENT
  nR_AreaMarkSensorOk             : INT := 10;  (*Area with the correct arrangement of the mark sensor [%]*)
END_VAR

VAR CONSTANT
  fC_MIN_CONVEYOR_SPEED           : REAL := 0.05;  (*[m/s]*)
END_VAR

(*EL1252*)
bI_Sensor1_State        := bIKp_CmdStartPrintSta;
tI_Sensor1_TimeStampPos := tIKp_TimeStampPos;
tI_Sensor1_TimeStampNeg := tIKn_TimeStampNeg;

IF bI_Reset THEN
	bL_inhibSensor1       := FALSE;
	bO_MarkDetected1      := FALSE;
	bL_S1_AcqOK           := FALSE;
END_IF;

(*zero divisions*)
IF    fI_Resolution = 0 THEN iL_Dbg_0Div := iL_Dbg_0Div + 1; RETURN;
ELSIF fI_MarkHeight = 0 THEN iL_Dbg_0Div := iL_Dbg_0Div + 1; RETURN;
END_IF;

iL_InhibitLength := FC_LREAL_TO_DINT((fI_SubstrateLength - fL_InhibitSubstrateDecrease) * (1 / (0.0254 / fI_Resolution)), pI_ConversionErr);
//bL_SpeedValid  := fI_ConveyorSpeed > fC_MIN_CONVEYOR_SPEED;
bL_SpeedValid    := bI_SpeedValid;


(* -------- Detection of rising edge on sensor1 --------*)
IF bI_Sensor1_State AND NOT bL_memS1_State AND NOT bL_inhibSensor1 AND bL_SpeedValid AND NOT bI_SimTriggerActive THEN
	tL_S1_RisingEdge := tI_Sensor1_TimeStampPos;

	IF bI_WithMark THEN					(*  if the paper is marked, *)
		bL_S1_AcqOK      := FALSE;(*  the function will wait until the falling edge to calculate the lateral offset too*)
	ELSE												(*  if the paper is not marked, *)
		bL_S1_AcqOK      := TRUE;	(*  the function will directly calculate the angle, can't calculate the lateral offset*)
		bL_inhibSensor1  := TRUE;
		bO_MarkDetected1 := TRUE;
	END_IF;

(* Calculate the current and sensor time stamp *)
	tL_CurrentTimeStamp  := F_GetCurDcTaskTime64();
	fL_CurrentTimeStamp  := (ULINT_TO_LREAL(tL_CurrentTimeStamp)     - (iI_CurrentTimeStampComp * 1_000)) / 1_000_000.0; (*in ms*)
	fI_Sensor1_TimeStamp := (ULINT_TO_LREAL(tI_Sensor1_TimeStampPos) - (iI_SensorTimeStampComp  * 1_000)) / 1_000_000.0; (*in ms*)

(* Treatment of the information *)
	fL_DeltaDistance := (fL_CurrentTimeStamp - fI_Sensor1_TimeStamp) * 0.001 * fI_ConveyorSpeed;	(* Distance in pulses that the substrate has traveled between the sensor detection and the PLC treatment *)
	fL_TempVar       := fL_DeltaDistance * (1 / (0.0254 / fI_Resolution));  (*1/1px*)	(* Travel of the substrate between the time of acquisition and the time of treatment *)
	iL_DeltaPosition := FC_LREAL_TO_DINT(fL_TempVar, pI_ConversionErr);
	iO_Offset_X0     := iI_CurrentPos - iL_DeltaPosition;	(* Position where the sheet has been detected *)
END_IF;

(*Debug & Test*)
IF bI_ManualTrigger AND bL_SpeedValid THEN
	bL_S1_AcqOK     := TRUE;
  bL_inhibSensor1 := TRUE;
  iO_Offset_X0    := iI_ManualTriggerPosition;	(* Position where the sheet has been detected *)
END_IF


(*debug - store max and minimal correction pulse*)
IF DINT_TO_UDINT(iL_DeltaPosition) > iL_DbgDeltaP_max THEN
	iL_DbgDeltaP_max := DINT_TO_UDINT(iL_DeltaPosition);
END_IF
IF DINT_TO_UDINT(iL_DeltaPosition) < iL_DbgDeltaP_min THEN
	iL_DbgDeltaP_min := DINT_TO_UDINT(iL_DeltaPosition);
END_IF


(* -------- Detection of falling edge, only for detection with mark --------*)
IF bI_WithMark AND NOT bI_Sensor1_State AND bL_memS1_State AND NOT bL_inhibSensor1 AND bL_SpeedValid AND NOT bI_SimTriggerActive THEN
	tL_S1_FallingEdge := tI_Sensor1_TimeStampNeg;
	fL_S1_Duration    := LREAL_TO_REAL(ULINT_TO_LREAL(tL_S1_FallingEdge) - ULINT_TO_LREAL(tL_S1_RisingEdge));		(* Calculate how long the signal was ON *)
	fL_S1_Length      := fL_S1_Duration * fI_ConveyorSpeed * 0.000_000_001;			(* Calculate the equivalence*)
	bL_S1_AcqOK       := TRUE;									(* now the function can continue to Angle & Offset calculation *)
	bL_inhibSensor1   := TRUE;
	bO_MarkDetected1  := TRUE;
END_IF;

bL_memS1_State := bI_Sensor1_State;			(* Memorization of the sensor1 state for next cycle *)


(*Check mark sensor detection*)
IF fI_ConveyorSpeed <> 0 THEN
  fb_TonCheckMarks(IN := (bL_SpeedValid AND NOT bL_S1_AcqOK), PT := REAL_TO_TIME((2 * fI_SubstrateLength) / fI_ConveyorSpeed * 1000) );
ELSE
  fb_TonCheckMarks(IN := FALSE);
END_IF


(* ------------ OFFSET CALCULATION ----------------- *)
IF bL_S1_AcqOK THEN
	IF bI_WithMark AND NOT bI_ManualTrigger THEN
    (*Sensor should aligned to the middle of the sensor (fI_MarkHeight / 2). *)
    (*With the difference of the measured lenght to the normal lenght, the fO_LateralOffset can be calculated*)
    (* invert in case of wrong mirrored marks *)
    IF bI_MarksInverted THEN
      fO_LateralOffset := -1*((fL_S1_Length * (fI_MarkHeight / 2 ) / (fI_MarkLength / 2)) - (fI_MarkHeight / 2 ));
    ELSE     
		  fO_LateralOffset := (fL_S1_Length * (fI_MarkHeight / 2 ) / (fI_MarkLength / 2)) - (fI_MarkHeight / 2 );
    END_IF
	ELSE
		fO_LateralOffset := 0;			(* if no mark on the paper, can't detect the offset *)
	END_IF;
	bL_S1_AcqOK  := FALSE;
	bO_StartTrig := TRUE;
ELSE
	bO_StartTrig := FALSE;
END_IF;


(*Check area with the correct arrangement of the mark sensor*)
nO_PrintMarkPosBits := 0;
IF fb_TonCheckMarks.Q THEN
  nO_PrintMarkPosBits.0 := TRUE; (*mark missing*) 
ELSE
  IF    (fO_LateralOffset = 0) 
     OR FC_COMPARE_RANGE_PERCENT( fI_ValueSet     := (fI_MarkHeight / 2)
                                , fI_ValueActual  := (fI_MarkHeight / 2) + fO_LateralOffset
                                , fI_RangePercent := nR_AreaMarkSensorOk)
  THEN 
    nO_PrintMarkPosBits.2 := TRUE; (*mark position in center*) 
  ELSIF fO_LateralOffset > 0 THEN
    nO_PrintMarkPosBits.1 := TRUE; (*mark position on side I*) 
  ELSIF fO_LateralOffset < 0 THEN
    nO_PrintMarkPosBits.3 := TRUE; (*mark position on side II*) 
  END_IF
END_IF


(*------------ start and stop signal treatment ------------*)

(*generate stop trigger*)
bL_StopCondition := (iI_CurrentPos >= (iO_Offset_X0 + iL_InhibitLength));
IF bL_StopCondition AND bL_inhibSensor1 THEN
	bL_inhibSensor1  := FALSE;
	bO_MarkDetected1 := FALSE;
END_IF;

END_FUNCTION_BLOCK

// ---- GlobalTextList.TcGTLO
TEXTLIST GlobalTextList
  10210 = '  x:%0.5f'
  6570 = '  y:%0.5f'
  781 = ' Camera offset Y [mm]: %f'
  2961 = ' cM: Camera start margin [m]: %f'
  5665 = ' Modus: %s'
  13668 = ' Nb teach marks: %d'
  13672 = ' Nb teach sectors: %d'
  9596 = ' Number of marks: %d'
  10437 = ' pW: Actual PrintUnit width [m]: %f'
  8296 = ' pWc: PrintUnit width [m]: %f'
  2948 = ' Sector of transmission: %d'
  5660 = ' Version number: %d'
  1184 = '%0.01f'
  14098 = '%0.02f'
  4085 = '%0.02f m/s'
  13676 = '%0.04f'
  8040 = '%0.06f'
  303 = '%0.0f'
  2502 = '%0.0f [m]'
  8178 = '%0.0f [px]'
  293 = '%0.1f'
  11885 = '%0.1f [cols]'
  430 = '%0.1f [m/min]'
  941 = '%0.1f [um]'
  10 = '%0.2f'
  993 = '%0.3f'
  1945 = '%0.3f [m/min]'
  6769 = '%0.3f [m/s]'
  4949 = '%0.3f [ms]'
  10891 = '%0.3f [m]'
  7216 = '%0.3f [px]'
  1864 = '%0.4f'
  11719 = '%0.4f  [m]'
  1796 = '%0.4f [ms]'
  7315 = '%0.4f [m]'
  1072 = '%0.5f'
  1822 = '%0.5f [m]'
  1887 = '%0.6f [m/s]'
  1147 = '%0.6f [ms]'
  820 = '%0.6f [m]'
  2289 = '%0.6f [um]'
  704 = '%1.1f'
  3079 = '%1.1f mm'
  3009 = '%1.1f mm/s'
  1930 = '%1.2f'
  741 = '%1.2f mm'
  3014 = '%1.3f mm'
  2489 = '%1.3f [mm]'
  6533 = '%1.3f [px]'
  3085 = '%1.4f m'
  7362 = '%1.4f [ms]'
  2560 = '%1.4f [m]'
  3481 = '%1.5f [m]'
  9 = '%d'
  3602 = '%d [px]'
  2955 = '%d [um]'
  456 = '%f'
  2383 = '%f [m/min]'
  5388 = '%f [mm]'
  812 = '%f [m]'
  2912 = '%f [s.p.min]'
  3959 = '%f [um]'
  27 = '%s'
  260 = '%s%%'
  9843 = '(Hw)Enable'
  3930 = '(not used) CameraToPrintUnit'
  17381 = '(viratual) generated'
  12232 = '*'
  447 = '+'
  7024 = '+/- %0.4f'
  8411 = '-'
  68 = '/'
  2589 = '1'
  2552 = '1. Activate (Drop)SpeedComp with Time set to 0\n\n2. Test print with production speed1\n   -> Measure displacement with Speed1\n\n3. Test print with production speed2\n   -> Measure displacement with Speed2\n\n4. Enter Speed and Displacement values in\n    table for Test1 and Test2\n\n5. Start new Time calculation'
  245 = '1. Activate (Drop)SpeedComp with Time set to 0\n\n2. Test print with Speed1\n   -> Measure displacement with Speed1\n\n3. Test print with Speed2\n   -> Measure displacement with Speed2\n\n4. Enter Speed and Displacement values in\n    table for Test1 and Test2\n\n5. Start new Time calculation'
  864 = '1. Activate (Drop)SpeedComp with Time set to 0\n\n2. Test1 print with production speed1\n   -> Measure displacement with Speed1\n\n3. Test2 print with production speed2\n   -> Measure displacement with Speed2\n\n4. Enter Speed and Displacement values in\n    table for Test1 and Test2\n\n5. Start new Time calculation'
  835 = '1. Activate (Drop)SpeedComp with Time set to 0\n\n2. Test1: print with production speed1\n   -> Measure displacement with Speed1\n\n3. Test2: print with production speed2\n   -> Measure displacement with Speed2\n\n4. Enter Speed and Displacement values in\n    table for Test1 and Test2\n\n5. Start new Time calculation'
  41 = '1. Activate DropSpeeCmp'
  1428 = '1. Activate DropSpeeComp\n   + Set Time to 0'
  1322 = '1. Activate DropSpeeComp\n   + Set Time to 0\n\n\n\n'
  1646 = '1. Activate DropSpeeComp\n   + Set Time to 0\n\n2. Test print with Speed1\n   + Measure displacement with Speed1\n\n'
  478 = '1. Activate DropSpeeComp\n   + Set Time to 0\n\n2. Test print with Speed1\n   + Measure displacement with Speed1\n\n3. Test print with Speed2\n   + Measure displacement with Speed2\n'
  2206 = '1. Activate DropSpeeComp\n   + Set Time to 0\n\n2. Test print with Speed1\n   + Measure displacement with Speed1\n\n3. Test print with Speed2\n   + Measure displacement with Speed2\n\n\n4. Enter values in table for Test1 and Test2\n\n5. Start new Time calculation'
  543 = '1. Activate DropSpeeComp\n   + Set Time to 0\n\n2. Test print with Speed1\n   + Measure displacement with Speed1\n\n3. Test print with Speed2\n   + Measure displacement with Speed2\n\n\n\n4. Enter values in table for Test1 and Test2'
  1417 = '1. Activate DropSpeeComp\n   + Set Time to 0\n\n2. Test print with Speed1\n   + Measure displacement with Speed1\n\n3. Test print with Speed2\n   + Measure displacement with Speed2\n\n5. Start new Time calculation\n\n4. Enter values in table for Test1 and Test2'
  2118 = '1. Activate DropSpeeComp\n   Set Time to 0'
  1160 = '1. Activate DropSpeeComp with Time set to 0\n\n2. Test print with Speed1\n   + Measure displacement with Speed1\n\n3. Test print with Speed2\n   + Measure displacement with Speed2\n\n\n4. Enter values in table for Test1 and Test2\n\n5. Start new Time calculation'
  1763 = '1. Activate DropSpeeComp with Time set to 0\n\n2. Test print with Speed1\n   + Measure displacement with Speed1\n\n3. Test print with Speed2\n   + Measure displacement with Speed2\n\n4. Enter values in table for Test1 and Test2\n\n5. Start new Time calculation'
  1928 = '1. Activate DropSpeeComp with Time set to 0\n\n2. Test print with Speed1\n   -> Measure displacement with Speed1\n\n3. Test print with Speed2\n   -> Measure displacement with Speed2\n\n4. Enter Speed and Displacement values\n     in table for Test1 and Test2\n\n5. Start new Time calculation'
  2230 = '1. Activate DropSpeeComp with Time set to 0\n\n2. Test print with Speed1\n   -> Measure displacement with Speed1\n\n3. Test print with Speed2\n   -> Measure displacement with Speed2\n\n4. Enter Speed and Displacement values in\n    table for Test1 and Test2\n\n5. Start new Time calculation'
  2617 = '1. Activate DropSpeeComp with Time set to 0\n\n2. Test print with Speed1\n   -> Measure displacement with Speed1\n\n3. Test print with Speed2\n   -> Measure displacement with Speed2\n\n4. Enter Speed and Displacement values in     table for Test1 and Test2\n\n5. Start new Time calculation'
  167 = '1. Activate DropSpeeComp with Time set to 0\n\n2. Test print with Speed1\n   -> Measure displacement with Speed1\n\n3. Test print with Speed2\n   -> Measure displacement with Speed2\n\n4. Enter Speed and Displacement values in table for Test1 and Test2\n\n5. Start new Time calculation'
  1944 = '1. Activate DropSpeeComp with Time set to 0\n\n2. Test print with Speed1\n   -> Measure displacement with Speed1\n\n3. Test print with Speed2\n   -> Measure displacement with Speed2\n\n4. Enter values in table for Test1 and Test2\n\n5. Start new Time calculation'
  363 = '1. Activate DropSpeedComp with Time set to 0\n\n2. Test print with Speed1\n   -> Measure displacement with Speed1\n\n3. Test print with Speed2\n   -> Measure displacement with Speed2\n\n4. Enter Speed and Displacement values in\n    table for Test1 and Test2\n\n5. Start new Time calculation'
  2048 = '1. Active DropSpeedComp'
  2104 = '1. Set Time to 0'
  7016 = '2*a'
  1505 = '2. Test print with Speed1\n   + Measure displacement with Speed1'
  2308 = '2. Test print with Speed1\n   Measure displacement with Speed1'
  1658 = '3. Test print with Speed2\n   + Measure displacement with Speed2'
  77 = '3. Test print with Speed2\n   Measure displacement with Speed2'
  550 = '4. Calculate new Time'
  581 = '4. Enter values in table for Test1 and Test2'
  1286 = '4. Start new Time calculation'
  2168 = '4p PLC'
  739 = '5. Start new Time calculation'
  8190 = '<'
  11083 = '<-'
  448 = '='
  6003 = '>'
  9654 = '>Camera(s)'
  1163 = '>FineAlignement'
  15769 = '>PrintPosition'
  18969 = '>WorkerPrint PG1 (Row1)'
  2212 = '>WorkerPrint PG2 (Row2)'
  19156 = 'a'
  14960 = 'a (mark size)'
  3758 = 'a/2'
  7335 = 'a: %d'
  4185 = 'Abort'
  3571 = 'Acknowledge'
  1383 = 'Act pos.'
  140 = 'Active'
  1300 = 'active camera device'
  517 = 'active camera device type'
  7324 = 'active camera mode'
  2160 = 'Actual Y-Resolution [dpi]: %1.4f'
  8699 = 'added points'
  1427 = 'ADS axis position'
  590 = 'ADS Axis Position'
  5009 = 'ADS command'
  717 = 'ADS Commands'
  9674 = 'ADS PG shift'
  2259 = 'ADS PU shift'
  4169 = 'ADS settings'
  723 = 'ADS Settings'
  15944 = 'All Epsitron'
  3353 = 'All Epsitron OK'
  5267 = 'All Inputs ok'
  5680 = 'AnalogMaxDigit'
  3775 = 'Auto'
  671 = 'AUTO/MANU CONTROL'
  4177 = 'Automatic Mode'
  1339 = 'Automatic or ManualTeach'
  2606 = 'AutomaticMode or ManualTeach'
  12039 = 'b'
  7246 = 'b (mark size)'
  9731 = 'B250'
  2262 = 'B254'
  16217 = 'B257'
  2111 = 'Back'
  608 = 'Bacl'
  3856 = 'bStopReady'
  210 = 'Busy'
  19400 = 'by calculation'
  6619 = 'C'
  411 = 'c'
  9048 = 'c (mark distance)'
  744 = 'C1'
  743 = 'C2'
  1065 = 'c: %d'
  3129 = 'c:%d'
  710 = 'Ca/Pu'
  136 = 'Calculate new time'
  1431 = 'Calculate new Time'
  13216 = 'Calender'
  6811 = 'cam simulation'
  1299 = 'Cam valid'
  1186 = 'Cam Valid'
  4259 = 'Camera'
  13991 = 'Camera activated'
  11573 = 'Camera Detail: %s'
  1141 = 'Camera ip address'
  1321 = 'camera mode desired'
  530 = 'camera mode desired (active cam)'
  1086 = 'Camera name'
  1061 = 'camera port'
  2103 = 'Camera sink'
  6170 = 'Camera temperature [°C]: %1.1f'
  5051 = 'Camera trigger'
  1990 = 'Camera type'
  9680 = 'Camera->PU'
  11139 = 'CameraToPrintUnit'
  8862 = 'CameraTrigger'
  14480 = 'CamPointsFifo'
  5607 = 'CamToPU'
  5019 = 'CanEx'
  7354 = 'cfb'
  10808 = 'Charged columns'
  8294 = 'Check delay'
  708 = 'Clean'
  3790 = 'Clean Active'
  719 = 'Clean after Capping'
  720 = 'Clean after Purge'
  1935 = 'Clean Head'
  1246 = 'Clean head (max %d)'
  711 = 'Clean Unit'
  15882 = 'Clean unit (max %d)'
  14428 = 'CleanCappPosition'
  4247 = 'CLEANER'
  4468 = 'Cleaner pump'
  265 = 'Cleaning'
  3760 = 'Cleaning Operations'
  740 = 'Cleaning Safe '
  4828 = 'CleaningProcess'
  212 = 'col'
  1396 = 'Column Precharge'
  6407 = 'Comp.'
  10565 = 'Compensation temperatur extension'
  11736 = 'configured camera mode, active=%s'
  10779 = 'Connected'
  9558 = 'constant'
  7336 = 'correction relative'
  6221 = 'csv'
  8478 = 'ct'
  3579 = 'CT'
  8221 = 'CT @Deformation (more corrections followed @Print!)'
  1165 = 'CT Id=%d'
  5554 = 'CT ImageDeformation'
  1850 = 'CT PrintRef'
  6824 = 'CT Status'
  17584 = 'CTDetail  @PrintWorker[1]  !No FineAlignment yet applied!'
  11030 = 'CTManager'
  15305 = 'Current'
  69 = 'current camera mode (active cam)'
  1219 = 'Current columen relative to Worker Attach'
  6060 = 'Current column'
  10240 = 'Current CT'
  10438 = 'Current position'
  10758 = 'Current reso used (from machine)'
  20158 = 'Current Speed'
  4981 = 'Current step'
  1573 = 'CurrentSpeed [m/s]'
  389 = 'D'
  2060 = 'Dead Time'
  1132 = 'Dead/Add Time'
  4013 = 'Dead/Add Time [ms]'
  21105 = 'Debug & Simulation'
  12899 = 'Deformation'
  1100 = 'DeformType'
  3003 = 'Delta P'
  2040 = 'Detect -> Cam'
  7545 = 'Detect -> Cam (Trig.Dist.)'
  18521 = 'Detected'
  6 = 'detected length [mm]'
  10000 = 'detected length [m]'
  1172 = 'Detected Marks: %d'
  9097 = 'Detection'
  10216 = 'Detection range [m]'
  12392 = 'DetectToCam'
  11747 = 'DetectToCamera'
  1597 = 'Device type'
  4990 = 'DevOpActive'
  5555 = 'Diff [mm]'
  8247 = 'Diff [m]'
  16644 = 'Direction'
  1171 = 'Disable left SLM'
  6432 = 'Disable right SLM'
  2162 = 'Displacement'
  1297 = 'Displacment'
  4696 = 'Distance in [p]'
  16193 = 'Distance [m]'
  4984 = 'DistBetweenMasks'
  3424 = 'DistToCamera'
  3798 = 'DO'
  152 = 'Done'
  1364 = 'Done LastMrk'
  4615 = 'DropSpeed'
  11858 = 'DropSpeed compensation'
  13254 = 'DropSpeed Compensation'
  1196 = 'DropSpeed Setup'
  4971 = 'DropSpeed [m/s]'
  3476 = 'DX'
  1038 = 'dx'
  8677 = 'dX (Global Deformation Shift)'
  1075 = 'dx (middle)'
  4842 = 'dX shift (points)'
  4026 = 'dx [mm]'
  6941 = 'dx [m]'
  15980 = 'dx:%0.5f'
  5761 = 'dx=%0.5f'
  1050 = 'DY'
  1039 = 'dy'
  10840 = 'dY (Global Deformation Shift)'
  2175 = 'dy [mm]'
  14658 = 'dy [m]'
  2520 = 'dy:%0.5f'
  15313 = 'dy=%0.5f'
  18481 = 'e state'
  2650 = 'Effective Encoder Resolution Detection'
  3372 = 'Effective[mm]'
  8187 = 'Effective[m]'
  5571 = 'Eject'
  4244 = 'Ejected'
  6817 = 'Ejected=1'
  2388 = 'EjectTriggerLength'
  3062 = 'EL7041'
  685 = 'EL7201'
  10657 = 'ElapsedTime: %s'
  4263 = 'Emergency stop'
  8 = 'Enable'
  2501 = 'Enable Correction'
  147 = 'Enable Speed Compensation'
  234 = 'Enabled'
  7765 = 'Enabled compensation'
  1980 = 'Encoder'
  7568 = 'Encoder Filter'
  4996 = 'encoder filter active'
  14488 = 'Encoder speed compensation factor'
  5880 = 'Encoder speed compensation reference speed'
  2208 = 'EncoderReso'
  9966 = 'EncoderResolution'
  6771 = 'EncSpeedCompFactor'
  9759 = 'EncSpeedCompRefSpeed'
  1636 = 'EncSpeedCorrection'
  417 = 'Endless'
  5930 = 'Engaged'
  714 = 'Enter Capping'
  688 = 'Epsitron Control'
  4621 = 'Err: %d'
  40 = 'Error'
  13934 = 'Error 0x%X'
  1158 = 'Error level'
  4543 = 'error: %d'
  731 = 'EStop'
  3722 = 'EStop Ok'
  4412 = 'exec'
  5028 = 'Exec'
  2082 = 'Execute device reset only in CU park position!'
  14686 = 'Execute device reset only in PU service position!'
  2569 = 'Execute device reset only in safe state'
  18335 = 'Exeeds max. speed=%f'
  11482 = 'Exhaust active'
  1734 = 'Exhaust system'
  2867 = 'Exhaust vacuum measurement 0-50mBar'
  715 = 'Exit Capping'
  3291 = 'Exporter'
  10708 = 'e_DeltaT'
  4278 = 'f (%d)'
  2541 = 'F=%d'
  1765 = 'Fast Stop Request'
  7021 = 'FastStop'
  1938 = 'Fault Acknowledge'
  11231 = 'Feature grid'
  17650 = 'FeatureGrid'
  4662 = 'feedback [mBar]'
  5376 = 'File Format'
  2633 = 'File Name'
  971 = 'File Path'
  3286 = 'filter active'
  682 = 'filter active (green)'
  12495 = 'Filter depth'
  1635 = 'filter=%d'
  2291 = 'Filters settings'
  705 = 'Force Close'
  9669 = 'Force DefGrid stream OFF'
  4095 = 'Force Grid OFF (gridPs=0)'
  729 = 'Force Open'
  12720 = 'ForceGrid OFF'
  3916 = 'Format'
  18523 = 'Format Machine'
  12999 = 'fPrintStartOffset'
  1948 = 'Frames for this image'
  1067 = 'From row: %d'
  913 = 'fsf'
  1148 = 'fsf\nsdfsd\nsdfsd'
  5979 = 'F[%d]'
  453 = 'Gap [mm]'
  1280 = 'Gap [m]'
  982 = 'Gap [m], %d [mm]'
  4929 = 'Global dX'
  1069 = 'Global dY'
  18887 = 'GlobalShift Dx/Dy'
  5637 = 'Grid Exporter'
  1397 = 'Grid ImageOffset Y [px]'
  12596 = 'Grid Points'
  7895 = 'Grid size c/r/y'
  851 = 'Grid Size X'
  1029 = 'Grid SizeY'
  6188 = 'GridPitch x/y'
  13281 = 'GridPoint history ->'
  15797 = 'GridPointsFifo'
  3068 = 'GridSel'
  5110 = 'h:%0.3f'
  15957 = 'h=%0.4f'
  5131 = 'Hardware'
  11305 = 'Head Gap [m]'
  5194 = 'Head Offset Plate [m]'
  1014 = 'History'
  12822 = 'Host: %s'
  2960 = 'HwEnable'
  388 = 'I'
  5854 = 'ID'
  1719 = 'id'
  18013 = 'Id'
  3111 = 'id of ct head'
  11673 = 'Idx'
  428 = 'Ign'
  597 = 'ignored'
  14585 = 'Image Height'
  9559 = 'Image Length'
  3696 = 'Image Length Job'
  425 = 'Image Width'
  2947 = 'ImageLength'
  4494 = 'ImageLength effect.'
  17474 = 'IMLen: %0.04f'
  12205 = 'IMWidth: %0.04f'
  733 = 'In     Out'
  6859 = 'InArea'
  9554 = 'Infeed'
  1262 = 'Inhibit trigger'
  15988 = 'Init'
  166 = 'Init ok'
  8950 = 'Initialized'
  9607 = 'InkQuantity'
  5070 = 'InPrintPos'
  3260 = 'Input (Fuse)'
  1115 = 'Inputs'
  3753 = 'Interlock'
  2159 = 'invalid & ignored marks'
  2281 = 'Invalid marks (ignored)'
  4159 = 'inverted'
  5409 = 'Inverted'
  6150 = 'inverted X'
  386 = 'Job'
  10238 = 'Job is active'
  1053 = 'JobActive'
  7197 = 'json'
  3174 = 'l'
  12184 = 'Len'
  2034 = 'Len Detect [mm]'
  2995 = 'Len Detected'
  8363 = 'LenghtMissmatch'
  3520 = 'Length check'
  18494 = 'Length Configured'
  14466 = 'Length diff'
  13542 = 'Length Effective'
  15936 = 'Length not in range'
  376 = 'Length [mm]'
  1522 = 'Length [m]'
  1876 = 'LenSq [mm]'
  267 = 'LenSq [m]'
  6355 = 'LenSquare'
  2735 = 'LenTr [mm]'
  14842 = 'LenTriangle'
  737 = 'LimitDN'
  4478 = 'Limits from machine'
  736 = 'LimitUP'
  15280 = 'LineCamera'
  18927 = 'Logger'
  11756 = 'LogLevel'
  8854 = 'Low intense mode'
  8103 = 'lsq=%0.4f'
  17552 = 'ltr=%0.4f'
  2934 = 'lx'
  2937 = 'ly'
  287 = 'm'
  3178 = 'm=%d'
  6479 = 'Machine Interface'
  1179 = 'MachineStopped'
  15 = 'Maintenance'
  3805 = 'MANU CONTROL'
  20108 = 'Manu Trigger'
  2076 = 'ManualTeach'
  539 = 'Mark at S1 invalid length'
  3844 = 'Mark at S1 too short'
  7032 = 'Mark at S2 invalid length'
  3478 = 'Mark at S2 too short'
  6031 = 'Mark Details'
  1296 = 'Mark History'
  1816 = 'Mark is flipped/inverted'
  15343 = 'Mark Lenght Margin'
  1191 = 'Mark length in [mm], minimum length=%0.02f [mm]'
  6077 = 'mark not proper detected'
  12613 = 'Mark per Use'
  9961 = 'Mark Settings'
  1952 = 'Mark teach'
  18681 = 'mark too short'
  16062 = 'MarkCamera'
  8898 = 'MarkDefinition'
  2476 = 'MarkDefinition Detail - Mark[%d]'
  20000 = 'MarkDetection'
  8025 = 'MarkDistFromCenter: %0.04f'
  9087 = 'marks valid'
  7504 = 'Master module idx'
  813 = 'MAV filter size "Dist in Pulse"'
  3301 = 'MAV filter size "Dist in Pulse" measured'
  12087 = 'MAV size "Dist in Pulse" measured'
  5710 = 'MAV size "Pulse Speed"'
  1189 = 'Max Limit'
  13601 = 'Max. Speed [m/s]'
  6002 = 'MaxMas'
  4885 = 'MaxMaster'
  516 = 'MaxModule'
  6815 = 'MaxPM'
  4790 = 'MaxSubstrate Factor'
  17117 = 'Measure: %d'
  12383 = 'MeasuredEncoderPulse'
  8147 = 'Measurement'
  19576 = 'Measurement aborted'
  12224 = 'measurement counter'
  22057 = 'Min Limit'
  16128 = 'Min. Speed'
  1173 = 'Min. Speed for Production'
  7865 = 'Min. speed production [m/min]'
  2019 = 'Min. Speed [m/s]'
  10619 = 'Min. Use Length'
  2528 = 'MinM'
  5381 = 'MinMa'
  6191 = 'MinMas'
  3216 = 'MinMaster'
  3134 = 'MinMstrer'
  2492 = 'MinProd'
  2310 = 'MinProd.'
  21567 = 'Mis'
  1193 = 'Missed'
  1120 = 'missed'
  1712 = 'missed mark'
  17989 = 'Missing'
  9496 = 'missing marks'
  4567 = 'mm'
  1855 = 'Mode'
  15104 = 'Mode: %s'
  4697 = 'mode=%d'
  7218 = 'Motion'
  1942 = 'MOTION'
  3737 = 'Move Done'
  3074 = 'Move Z axis down after cleaning'
  2526 = 'Moving'
  5512 = 'Moving > Min.Speed for production'
  1914 = 'Name'
  10904 = 'Nbr Marks'
  1164 = 'Nbr Uses'
  13510 = 'No'
  17976 = 'no'
  784 = 'node'
  13171 = 'normal'
  16031 = 'Normal'
  1861 = 'Not all frames contain teach p'
  875 = 'Not all frames contain teach points'
  3138 = 'not engaged (Service)'
  11 = 'Not enough teach points for mode'
  2433 = 'NOTE: might be setup internally'
  10357 = 'num of grid points for job'
  1860 = 'num: %d'
  1919 = 'number exports, max:100'
  4362 = 'number of attached cts'
  385 = 'NumCTs'
  7300 = 'O'
  4393 = 'Off delay'
  5911 = 'OK'
  1847 = 'Open Shutter'
  511 = 'OPERATIONS'
  12010 = 'OtherMarks'
  1406 = 'Out Dir'
  2788 = 'Out Path'
  13228 = 'Outlet'
  5862 = 'OutputPath'
  2864 = 'Outside of machine'
  2527 = 'P\n%s'
  1774 = 'P%d'
  7846 = 'P1'
  18520 = 'P2'
  16371 = 'P3'
  2574 = 'P4'
  3836 = 'p: %d'
  1868 = 'PA'
  1923 = 'pA'
  11770 = 'PA1 WorkerPos'
  709 = 'Park'
  4056 = 'ParkPosition'
  1926 = 'pB'
  4279 = 'Permanent activation'
  1283 = 'PG '
  12785 = 'PG enable'
  3101 = 'PG XPosition'
  3591 = 'PG XPosition [m]'
  6193 = 'PG XPosition [um]'
  500 = 'PG1'
  501 = 'PG2'
  1192 = 'PG: %s'
  3020 = 'Place'
  1169 = 'PM'
  5877 = 'PM Distance to prev PM [m]'
  2049 = 'PM Distance to prev. PM [m]'
  336 = 'PM Distance to previvous PM [m]'
  20630 = 'PM in maintenance position'
  18050 = 'PM in printing position'
  2652 = 'PM Pos mech. to current Master'
  2540 = 'PM Pos mech. to current Master PU'
  9645 = 'PM position'
  2884 = 'PM position on main tracker'
  327 = 'PM position to prev'
  4663 = 'PM position to previous'
  18635 = 'PM X to Master Distance [m]'
  1121 = 'PmPosition=%0.5f   NOTE: PmPosition might be setup/added internally'
  5363 = 'Points'
  8746 = 'Port: %s'
  21704 = 'Pos'
  401 = 'Position'
  3032 = 'Position A'
  3038 = 'Position B'
  3044 = 'Position p1'
  3050 = 'Position p2'
  4232 = 'Position p3'
  4240 = 'Position p4'
  4208 = 'Position [mm]'
  7104 = 'Position [m]'
  8615 = 'Position [SubPx]'
  4770 = 'POSITIONS'
  1116 = 'Pre-StartOffset'
  566 = 'Pre-StartShiftFactor'
  2951 = 'Pre-StartShiftOffset'
  2554 = 'PreStart'
  5281 = 'PreStart (Factor/Offset)'
  7030 = 'PreStart ShiftFactor'
  5299 = 'PreStart ShiftOffset'
  10387 = 'PRG_PRINT'
  164 = 'Print'
  738 = 'Print '
  1180 = 'Print Direction (1=reverse)'
  14325 = 'Print enabled'
  1049 = 'Print Position'
  734 = 'Print Unit'
  4516 = 'Print unit (max %d)'
  12625 = 'Print1'
  3057 = 'Print2'
  5115 = 'Printhead 1'
  3223 = 'Printhead 2'
  8129 = 'PrintModule'
  18556 = 'PrintOffsetX'
  3350 = 'PrintOffsetY'
  10191 = 'PrintON'
  1536 = 'PrintPosition'
  4542 = 'PrintResolution'
  529 = 'PrintSpeed'
  4012 = 'PrintUnit temp at calibration [°C]: %1.1f'
  2680 = 'PrintUnit temperature [°C]: %1.1f'
  2360 = 'processed grid points'
  11146 = 'Produced: %s'
  5301 = 'ProductionSpeed'
  5878 = 'PU'
  4979 = 'PU 4p correction'
  2391 = 'PU 4p correction PLC'
  7392 = 'PU 4p correction PUC'
  6196 = 'PU banana correction'
  18230 = 'Pulse from encoder'
  21913 = 'Pulse Speed'
  8792 = 'Pump set [%]'
  593 = 'Purge'
  721 = 'Purge after Capping'
  13588 = 'PuToWorker'
  4094 = 'PyBusy'
  1213 = 'PyDefDone'
  12566 = 'PyError'
  2980 = 'PyId'
  11014 = 'PyPos'
  11517 = 'Python'
  1054 = 'Python Interface'
  10985 = 'PyUpd'
  90 = 'R'
  1066 = 'r: %d'
  7744 = 'r:%d'
  6096 = 'reached'
  150 = 'Ready'
  703 = 'Ref'
  11729 = 'reference'
  468 = 'Refresh'
  1058 = 'Reg.Points'
  3463 = 'Release from machine'
  1292 = 'Repeat History'
  3912 = 'RepeatLength'
  2586 = 'Reset'
  7014 = 'Reverse'
  4287 = 'Reverse cleaning drive'
  1181 = 'Reverse Direction'
  1955 = 'row'
  13758 = 'Rows: %d'
  4445 = 'Run down delay'
  3142 = 'Running'
  2929 = 'rx'
  10078 = 'RxCtr'
  2932 = 'ry'
  407 = 'S'
  5317 = 's'
  5767 = 's: %d'
  3768 = 'Safe Running Condition'
  3745 = 'Safety'
  17962 = 'Safety cover'
  15672 = 'Safety doors'
  8652 = 'Safety ok'
  3730 = 'SafetyConditionOK'
  3186 = 'Save CT'
  12285 = 'scanned points'
  19355 = 'Scrap:    %s'
  8666 = 'Script alive'
  6352 = 'Sector msg'
  7047 = 'Sel PH : %d '
  6555 = 'Selected for printing'
  14908 = 'Selection MasterModule'
  5838 = 'Send Loop test message'
  3413 = 'Sensor detect errors'
  742 = 'Serv'
  3783 = 'Service'
  2692 = 'ServiceEnabled'
  4356 = 'Set'
  1665 = 'Set value'
  5081 = 'Setpoint #1 [%]'
  2548 = 'Setpoint #2 [%]'
  1673 = 'Setpoint #3 [%]'
  3808 = 'Setpoint #4 [%]'
  2275 = 'Setpoint intensity'
  4255 = 'Setpoint [%]'
  61 = 'Settings'
  14005 = 'Setup'
  1795 = 'Setup new Time'
  308 = 'Setup SpeedCompensation'
  986 = 'Setup [mm]'
  21074 = 'Setup [m]'
  5118 = 'Sh'
  15331 = 'Sheet detect supervision'
  2258 = 'SheetCycle'
  1382 = 'SheetDetect'
  3305 = 'SheetGap'
  2344 = 'SheetGap [mm]'
  1697 = 'SheetLength'
  2532 = 'SheetLength [mm]'
  822 = 'SheetSpeed'
  1118 = 'SheetSpeed [m/min]'
  2238 = 'SheetTrigger'
  5168 = 'ShiftFact'
  6358 = 'ShiftOffs'
  6611 = 'Show Details'
  21803 = 'Show PC'
  20887 = 'Show PH'
  727 = 'Shutter'
  1344 = 'Sim'
  5078 = 'Sim MarkCamera'
  18626 = 'Sim MarkDetection'
  10659 = 'Sim Module'
  5898 = 'Sim position'
  2393 = 'Sim Position %0.3f [m/s]'
  12400 = 'simulate'
  11236 = 'Simulation'
  450 = 'Simulation auto-trigger'
  159 = 'Simulation enable'
  3368 = 'simulation mode'
  19662 = 'Specific Modules'
  2330 = 'Speed'
  6688 = 'speed compensationa active'
  10686 = 'Speed Exceeded'
  15504 = 'Speed m/min'
  181 = 'Speed m/s'
  2930 = 'Speed valid'
  105 = 'Speed [m/min]'
  1484 = 'Speed [m/min] %0.03f [m/s]'
  37 = 'Speed [m/min] %0.03s [m/s]'
  1515 = 'Speed [m/min] %s [m/s]'
  12089 = 'Speed [m/s]'
  1654 = 'Speed [sheet/h]'
  1220 = 'SpeedComp'
  18209 = 'SpeedExeeded'
  3813 = 'SPEEDS'
  12942 = 'sq:%0.3f'
  2356 = 'square length [mm]'
  12697 = 'square length [m]'
  1229 = 'St'
  4781 = 'Standby'
  5000 = 'Start Cleaning'
  20519 = 'start overrun'
  8343 = 'Start overrun'
  508 = 'Start Purge'
  4358 = 'Start up offset'
  9434 = 'start update'
  8070 = 'Started'
  14044 = 'StartMark'
  1620 = 'StartOffs'
  1680 = 'State'
  7664 = 'State name'
  18 = 'Status'
  3715 = 'STATUS'
  12536 = 'Step'
  12315 = 'Stop'
  2267 = 'Stop -> 0 [m/s]'
  17146 = 'Stop Request'
  5135 = 'SubPx'
  9498 = 'Substrate Gap (sim)'
  806 = 'Substrate Length'
  11702 = 'Substrate Width'
  3446 = 'SubstrateLength'
  1519 = 'SubstrateLength effect.'
  687 = 'SystemReady'
  5130 = 't: %d'
  4402 = 'Target'
  9116 = 'Target speed'
  5478 = 'Target speed reached'
  1960 = 'TargetSpeed [m/s]'
  11241 = 'TcpIpClient'
  5655 = 'Teach'
  15269 = 'teached marks'
  19842 = 'Teached Marks: %d'
  2734 = 'teached points'
  21 = 'TeachP'
  460 = 'TeachPoints first frame'
  1422 = 'TeachPoints in first frame'
  10982 = 'Temp at calibration [°C]: %1.1f'
  62 = 'Test'
  4175 = 'TEst'
  2921 = 'Test mode!'
  1251 = 'Test1'
  2109 = 'Test2'
  122 = 'Time'
  8956 = 'To row: %d'
  14553 = 'TODO'
  1520 = 'Tolerance'
  5472 = 'too long'
  3304 = 'too long$'
  8448 = 'Too short'
  3182 = 'too short'
  5716 = 'Total columns'
  7951 = 'tr:%0.3f'
  5292 = 'TrackPos'
  3091 = 'triangle length [mm]'
  16029 = 'triangle length [m]'
  7998 = 'Trigger active'
  228 = 'Trigger Armed'
  2681 = 'TriggerDistance'
  1388 = 'TriggerPulseLength'
  13192 = 'TrigToCam'
  7368 = 'T_PL1'
  1074 = 'T_PL2'
  11769 = 'update done'
  1306 = 'Use Global Grid Shift'
  5046 = 'UseCameraTrigger'
  10877 = 'UseCameraTriggerFeedback'
  5635 = 'UseLength'
  18311 = 'UsePerRepeat'
  3104 = 'v'
  5948 = 'V'
  4271 = 'VACUUM'
  4759 = 'Vacuum pump'
  2945 = 'valid'
  2158 = 'vbn'
  12744 = 'Verbose'
  1735 = 'Verbose mode'
  745 = 'Wait'
  746 = 'Waiting'
  4224 = 'Warning level'
  11338 = 'With Mark'
  3026 = 'Work'
  9075 = 'Worker enable'
  18138 = 'Worker PrintEnable'
  19928 = 'WorkerCamera'
  15457 = 'WorkercCamera'
  13015 = 'WorkerDeform'
  4305 = 'WorkerDeformation'
  11590 = 'WorkerDelete'
  2580 = 'WorkerOffset'
  670 = 'WorkerOffset (PU/PM/PG)'
  1622 = 'WorkerPos (Attach)'
  12 = 'WorkerPos (to Master PM)'
  7284 = 'WorkerPosition'
  13745 = 'WorkerPrint %s'
  8780 = 'WorkerPrint enable'
  2559 = 'WorkerPrint1'
  6462 = 'WorkerPrint1 Line1'
  2497 = 'WorkerPrint2'
  14277 = 'WorkerPrint[1]'
  13424 = 'WorkerPrint[2]'
  6175 = 'WorkerPrint_fPrintStartOffset'
  6394 = 'WorkerPython'
  2890 = 'WorkerVerify'
  3090 = 'Working  pCT'
  2940 = 'x'
  9460 = 'X Ref'
  12401 = 'x [px 4800dpi]'
  886 = 'X0'
  15726 = 'X0 [SubPx]'
  15794 = 'X0: %d'
  4503 = 'x=%0.4f'
  17127 = 'XD: %d'
  887 = 'XS'
  194 = 'XS (+offset + Corrections X)'
  10930 = 'x_P [mm]'
  3312 = 'x_ref'
  14137 = 'x_ref_P [mm]'
  2942 = 'y'
  1070 = 'y [px 4800dpi]'
  8833 = 'Y-Resolution at calibration [dpi]: %1.4f'
  1 = 'y-shift'
  4527 = 'y=%0.4f'
  9660 = 'Yes'
  2488 = 'yes'
  5240 = 'y_max'
  1071 = 'y_P [mm]'
  10734 = 'y_ref'
  7467 = 'y_ref_P [mm]'
  2747 = 'Z Axis'
  1073 = '[%s]'
  13426 = '[-] WebStrech calculated'
  5404 = '[1] CT Id=%d'
  1166 = '[2] CT Id=%d'
  17264 = '[m/s] Max. Speed'
  11491 = '[m/s] Speed'
  3807 = '[mm/C]'
  1135 = '[mm]'
  4403 = '[m]'
  3395 = '[m] HeadGap'
  19619 = '[m] LateralRegister'
  8220 = '[m] Module2ToModule3'
  18328 = '[m] SubstrateLength'
  19359 = '[m] SubstrateThickness'
  2475 = '[p/um] Encoder resolution'
  17520 = '[um] SubstrateThickness'
  3480 = '^'
END_TEXTLIST

// ---- POUs/Machine/CleaningStation/_VISU_CleanCH.TcVIS
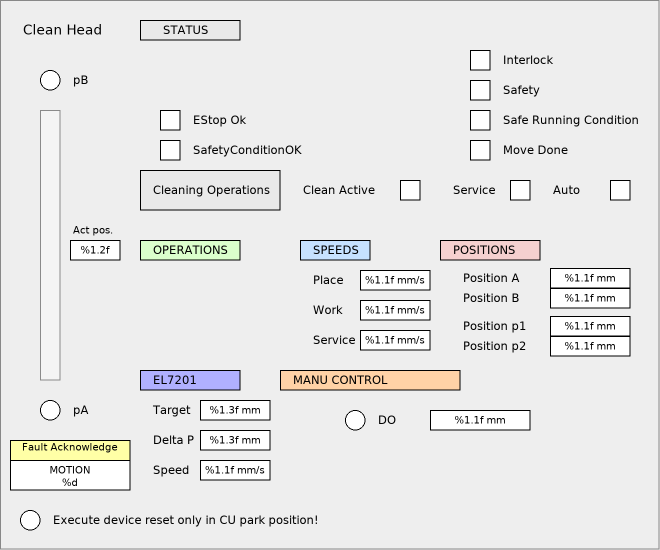
VISUALIZATION _VISU_CleanCH  // 660x550
VAR_IN_OUT
  mInst  : FB_CleaningMotorAxisCH;
END_VAR
    Rectangle (0,0 660x550)
    Polyline (210,380)
    Polyline (510,250)
    Polyline (300,250)
    Rectangle (280,370 180x20)
    Rectangle (300,240 70x20)
    Rectangle (440,240 100x20)
    Rectangle (140,240 100x20)
    Rectangle (70,400 40x20), "pA"
    Ellipse (40,400 20x20), colour toggle: mInst.bL_Sensor_pA
    Ellipse (40,70 20x20), colour toggle: mInst.bI_Sensor_pB
    Rectangle (70,70 50x20), "pB"
    Rectangle (70,240 50x20), "%1.2f", text variable: 1000 * mInst.fB_Axis.fO_ActualPosition
    Rectangle (375,410 40x20), "DO"
    Rectangle (290,370 170x20), "MANU CONTROL"
    Polyline (450,380)
    Rectangle (310,240 70x20), "SPEEDS"
    Rectangle (360,270 70x20), "%1.1f mm/s", text variable: mInst.sI_SpeedDef.fP_PlaceSpeed
        OnMouseDown: write the text variable via VisuDialogs.Numpad
    Rectangle (360,300 70x20), "%1.1f mm/s", text variable: mInst.sI_SpeedDef.fP_WorkSpeed
        OnMouseDown: write the text variable via VisuDialogs.Numpad
    Rectangle (360,330 70x20), "%1.1f mm/s", text variable: mInst.sI_SpeedDef.fP_ServiceSpeed
        OnMouseDown: write the text variable via VisuDialogs.Numpad
    Rectangle (310,270 60x20), "Place"
    Rectangle (310,300 60x20), "Work"
    Rectangle (310,330 60x20), "Service"
        OnMouseDown: write the text variable via Edit
    Rectangle (550,268 80x20), "%1.1f mm", text variable: mInst.fI_Position_A
        OnMouseDown: write the text variable via VisuDialogs.Numpad
    Rectangle (460,268 85x20), "Position A"
    Rectangle (460,288 85x20), "Position B"
    Rectangle (550,288 80x20), "%1.1f mm", text variable: mInst.fI_Position_B
        OnMouseDown: write the text variable via VisuDialogs.Numpad
    Rectangle (450,240 90x20), "POSITIONS"
    Polyline (210,250)
    Rectangle (150,240 90x20), "OPERATIONS"
    Scrollbar (40,110 20x270)
        p3598130195: mInst.sADS_CleanAxis.sO_AxisPosition.fC_Min
        p2245068023: mInst.sADS_CleanAxis.sO_AxisPosition.fC_Max
        p1057716461: mInst.fB_Axis.fO_ActualPosition * 1000
    Ellipse (345,410 20x20), colour toggle: mInst.sADS_CleanAxis.bI_ManualMove, input disabled if: NOT mInst.sADS_CleanAxis.bO_ManualMoveCanEx
        toggle mInst.sADS_CleanAxis.bI_ManualMove
    Rectangle (20,20 120x20), "Clean Head"
    Rectangle (140,370 100x20)
    Rectangle (150,460 70x20), "Speed"
    Rectangle (200,460 70x20), "%1.1f mm/s", text variable: 1000 * mInst.fB_Axis.fI_SpeedLimit
    Rectangle (150,370 90x20), "EL7201"
    Rectangle (10,440 120x50), "Fault Acknowledge", colour toggle: (mInst.wL_ErrorCode) <> 0
    Polyline (130,450)
    RoundedRectangle (10,460 120x30), "%d", text variable: mInst.wL_ErrorCode
        tap mInst.sADS_CleanAxis.bI_FaultAck
    RoundedRectangle (40,460 60x20), "MOTION"
    Rectangle (140,170 140x40)
    Rectangle (140,20 100x20)
    Polyline (140,30)
    Polyline (240,30)
    Rectangle (160,20 60x20), "STATUS"
    RoundedRectangle (160,110 20x20), colour toggle: NOT mInst.bI_Emergency
    RoundedRectangle (160,140 20x20), colour toggle: mInst.bI_SafetyOk
    RoundedRectangle (470,140 20x20), colour toggle: NOT mInst.bL_Busy
    Rectangle (190,110 120x20), "EStop Ok"
    Rectangle (190,140 120x20), "SafetyConditionOK"
    Rectangle (500,140 90x20), "Move Done"
    RoundedRectangle (470,80 20x20), colour toggle: mInst.bI_SafeToMove
    Rectangle (500,80 120x20), "Safety"
    RoundedRectangle (470,50 20x20), colour toggle: mInst.bI_SafeToMove
    Rectangle (500,50 120x20), "Interlock"
    Polyline (650,160)
    Rectangle (150,180 140x20), "Cleaning Operations"
    Polyline (280,200)
    RoundedRectangle (470,110 20x20), colour toggle: mInst.bL_SafeRunningCondition
    Rectangle (500,110 150x20), "Safe Running Condition"
    RoundedRectangle (610,180 20x20), colour toggle: mInst.bI_UsrAutoMode
    Rectangle (550,180 60x20), "Auto"
    Polyline (350,80)
    RoundedRectangle (510,180 20x20), colour toggle: mInst.bI_UsrService
    Rectangle (450,180 60x20), "Service"
    Rectangle (300,180 90x20), "Clean Active"
    RoundedRectangle (400,180 20x20), colour toggle: mInst.bI_DevOpActive
    Rectangle (200,400 70x20), "%1.3f mm", text variable: 1000 * mInst.fB_Axis.fI_TargetPosition
    Rectangle (150,400 70x20), "Target"
    Rectangle (150,430 70x20), "Delta P"
    Rectangle (200,430 70x20), "%1.3f mm", text variable: 1000 * mInst.fB_Axis.fL_Delta_P
    Rectangle (430,410 100x20), "%1.1f mm", text variable: mInst.sADS_CleanAxis.fI_ManualTargetPos
        OnMouseDown: write the text variable via VisuDialogs.Numpad, min mInst.fI_Position_A, max mInst.fI_Position_B
    Rectangle (550,316 80x20), "%1.1f mm", text variable: mInst.fI_Position_p1
        OnMouseDown: write the text variable via VisuDialogs.Numpad
    Rectangle (460,316 85x20), "Position p1"
    Rectangle (460,336 85x20), "Position p2"
    Rectangle (550,336 80x20), "%1.1f mm", text variable: mInst.fI_Position_p2
        OnMouseDown: write the text variable via VisuDialogs.Numpad
    Ellipse (20,510 20x20), colour toggle: mInst.bIDp_DeviceReset, input disabled if: NOT mInst.bI_CUinPosCappingClean
        tap mInst.bIDp_DeviceReset
    Rectangle (50,510 306x20), "Execute device reset only in CU park position!"
    Rectangle (70,220 50x20), "Act pos."
END_VISUALIZATION

// ---- POUs/Machine/CleaningStation/_VISU_CleanCU.TcVIS
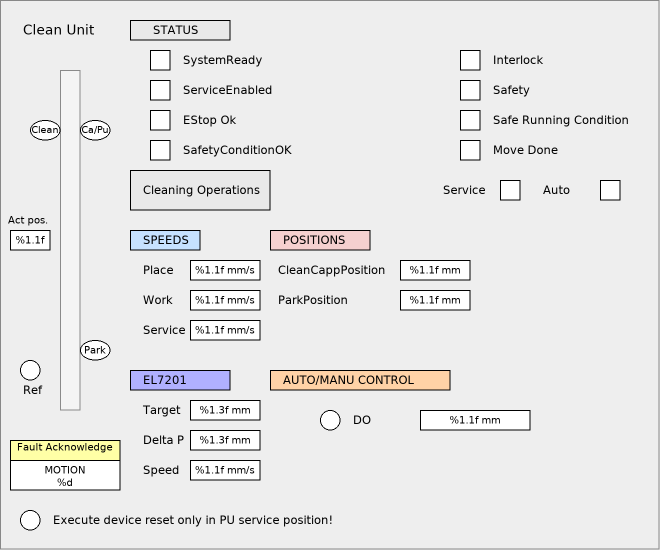
VISUALIZATION _VISU_CleanCU  // 660x550
VAR_IN_OUT
  mInst  : FB_CleaningMotorAxisCU;
END_VAR
    Rectangle (0,0 660x550)
    Polyline (200,380)
    Rectangle (130,370 100x20)
    Rectangle (270,370 180x20)
    Rectangle (270,230 100x20)
    Rectangle (130,230 70x20)
    Rectangle (280,370 170x20), "AUTO/MANU CONTROL"
    Polyline (440,380)
    Ellipse (20,360 20x20), colour toggle: mInst.bL_ReferenceSensor
    Rectangle (20,380 30x20), "Ref"
    Scrollbar (60,70 20x340)
        p3598130195: -0.01
        p2245068023: 0.6
        p1057716461: mInst.fB_Axis.fO_ActualPosition
    Rectangle (10,230 40x20), "%1.1f", text variable: 1000 * mInst.fB_Axis.fO_ActualPosition
    Rectangle (140,230 70x20), "SPEEDS"
    Polyline (130,240)
    Polyline (340,240)
    Rectangle (280,230 90x20), "POSITIONS"
    Rectangle (190,400 70x20), "%1.3f mm", text variable: 1000 * mInst.fB_Axis.fI_TargetPosition
    Rectangle (140,400 70x20), "Target"
    Rectangle (140,460 70x20), "Speed"
    Rectangle (190,460 70x20), "%1.1f mm/s", text variable: 1000 * mInst.fB_Axis.fI_SpeedLimit
    Rectangle (140,370 90x20), "EL7201"
    Rectangle (140,430 70x20), "Delta P"
    Rectangle (190,430 70x20), "%1.3f mm", text variable: 1000 * mInst.fB_Axis.fL_Delta_P
    Ellipse (30,120 30x20), "Clean", colour toggle: mInst.pInPosCappingClean
    Ellipse (80,340 30x20), "Park", colour toggle: mInst.pInPosPark
    Ellipse (80,120 30x20), "Ca/Pu", colour toggle: mInst.pInPosCappingClean
    Rectangle (20,20 110x20), "Clean Unit"
    Rectangle (10,440 110x50), "Fault Acknowledge", colour toggle: (mInst.wL_ErrorCode) <> 0
    RoundedRectangle (10,460 110x30), "%d", text variable: mInst.wL_ErrorCode
        tap mInst.sADS_CleanAxis.bI_FaultAck
    RoundedRectangle (10,460 110x20), "MOTION"
    Rectangle (130,170 140x40)
    Rectangle (130,20 100x20)
    Polyline (130,30)
    Polyline (230,30)
    Rectangle (150,20 60x20), "STATUS"
    RoundedRectangle (150,80 20x20), colour toggle: mInst.bI_UsrService
    RoundedRectangle (150,110 20x20), colour toggle: NOT mInst.bI_Emergency
    RoundedRectangle (150,140 20x20), colour toggle: mInst.bI_SafetyOk
    RoundedRectangle (460,140 20x20), colour toggle: NOT mInst.bL_Busy
    RoundedRectangle (150,50 20x20), colour toggle: mInst.bI_MachineReady
    Rectangle (180,50 120x20), "SystemReady"
    Rectangle (180,80 120x20), "ServiceEnabled"
    Rectangle (180,110 120x20), "EStop Ok"
    Rectangle (180,140 120x20), "SafetyConditionOK"
    Rectangle (490,140 90x20), "Move Done"
    RoundedRectangle (460,80 20x20), colour toggle: mInst.bI_SafeToMove
    Rectangle (490,80 120x20), "Safety"
    RoundedRectangle (460,50 20x20), colour toggle: mInst.bI_SafeToMove
    Rectangle (490,50 120x20), "Interlock"
    Polyline (640,160)
    Rectangle (140,180 140x20), "Cleaning Operations"
    Polyline (270,200)
    RoundedRectangle (460,110 20x20), colour toggle: mInst.bL_SafeRunningCondition
    Rectangle (490,110 150x20), "Safe Running Condition"
    RoundedRectangle (600,180 20x20), colour toggle: mInst.bI_UsrAutoMode
    Rectangle (540,180 60x20), "Auto"
    Polyline (340,80)
    RoundedRectangle (500,180 20x20), colour toggle: mInst.bI_UsrService
    Rectangle (440,180 60x20), "Service"
    Rectangle (420,410 110x20), "%1.1f mm", text variable: mInst.sADS_CleanAxis.fI_ManualTargetPos
        OnMouseDown: write the text variable via VisuDialogs.Numpad, min mInst.sADS_CleanAxis.sO_AxisPosition.fC_Min, max mInst.sADS_CleanAxis.sO_AxisPosition.fC_Max
    Rectangle (350,410 60x20), "DO"
    Ellipse (320,410 20x20), colour toggle: mInst.sADS_CleanAxis.bI_ManualMove, input disabled if: NOT mInst.sADS_CleanAxis.bO_ManualMoveCanEx
        toggle mInst.sADS_CleanAxis.bI_ManualMove
    Rectangle (190,260 70x20), "%1.1f mm/s", text variable: mInst.sI_SpeedDef.fP_PlaceSpeed
        OnMouseDown: write the text variable via VisuDialogs.Numpad
    Rectangle (190,290 70x20), "%1.1f mm/s", text variable: mInst.sI_SpeedDef.fP_WorkSpeed
        OnMouseDown: write the text variable via VisuDialogs.Numpad
    Rectangle (190,320 70x20), "%1.1f mm/s", text variable: mInst.sI_SpeedDef.fP_ServiceSpeed
        OnMouseDown: write the text variable via VisuDialogs.Numpad
    Rectangle (140,260 60x20), "Place"
    Rectangle (140,290 60x20), "Work"
    Rectangle (140,320 60x20), "Service"
    Rectangle (400,260 70x20), "%1.1f mm", text variable: mInst.fI_PositionCappingClean
        OnMouseDown: write the text variable via VisuDialogs.Numpad
    Rectangle (275,260 125x20), "CleanCappPosition"
    Rectangle (400,290 70x20), "%1.1f mm", text variable: mInst.fI_PositionPark
        OnMouseDown: write the text variable via VisuDialogs.Numpad
    Rectangle (275,290 125x20), "ParkPosition"
    Ellipse (20,510 20x20), colour toggle: mInst.bIDp_DeviceReset, input disabled if: mInst.bI_PUinPosService
        tap mInst.bIDp_DeviceReset
    Rectangle (50,510 306x20), "Execute device reset only in PU service position!"
    Rectangle (5,210 50x20), "Act pos."
END_VISUALIZATION

// ---- POUs/Machine/CleaningStation/_VISU_CleanProcess.TcVIS
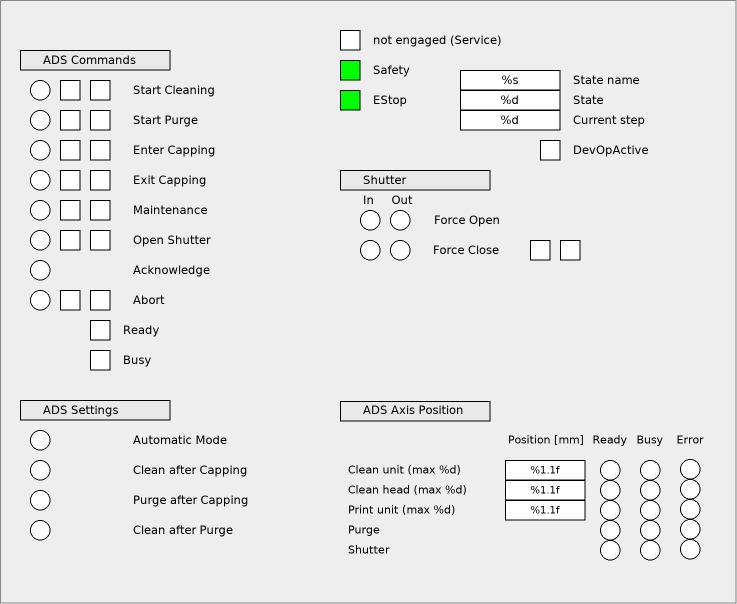
VISUALIZATION _VISU_CleanProcess  // 737x604
VAR_IN_OUT
  mInst            : FB_CleaningProcess;
  mInst_AdsProcess : FB_ADS_CleanProcess;
  mInst_AdsCU      : FB_ADS_CleanAxis;
  mInst_AdsCH      : FB_ADS_CleanAxis;
  mInst_AdsPU      : FB_ADS_CleanAxis;
  mInst_AdsPurge   : FB_ADS_CleanAxis;
  _bShutterExist   : BOOL;
  mInst_AdsShutter : FB_ADS_CleanAxis;
  mInst_FbShutter  : FB_SHUTTER;
END_VAR
    Rectangle (0,0 737x604)
    Polyline (20,50)
    Polyline (360,360)
    Rectangle (130,80 90x20), "Start Cleaning"
    Ellipse (30,80 20x20), colour toggle: mInst_AdsProcess.bI_Clean
        tap mInst_AdsProcess.bI_Clean
    Rectangle (130,110 90x20), "Start Purge"
    Rectangle (130,140 90x20), "Enter Capping"
    Rectangle (130,170 90x20), "Exit Capping"
    Rectangle (130,200 90x20), "Maintenance"
    RoundedRectangle (90,320 20x20), colour toggle: mInst_AdsProcess.bO_Ready
    Rectangle (120,320 120x20), "Ready"
    Rectangle (460,70 100x20), "%s", text variable: mInst.sL_CurrentState^.sL_StateName
    Rectangle (570,70 100x20), "State name"
    Rectangle (460,90 100x20), "%d", text variable: mInst.sL_CurrentState^.iL_State
    Rectangle (570,90 100x20), "State"
    Rectangle (20,50 150x20)
    Rectangle (40,50 130x20), "ADS Commands"
    RoundedRectangle (60,80 20x20), colour toggle: mInst_AdsProcess.bO_CleanCanEx
    RoundedRectangle (90,80 20x20), colour toggle: mInst_AdsProcess.bO_CleanExec
    Ellipse (30,110 20x20), colour toggle: mInst_AdsProcess.bI_Purge
        tap mInst_AdsProcess.bI_Purge
    RoundedRectangle (60,110 20x20), colour toggle: mInst_AdsProcess.bO_PurgeCanEx
    RoundedRectangle (90,110 20x20), colour toggle: mInst_AdsProcess.bO_PurgeExec
    Ellipse (30,140 20x20), colour toggle: mInst_AdsProcess.bI_StartCapping
        tap mInst_AdsProcess.bI_StartCapping
    RoundedRectangle (60,140 20x20), colour toggle: mInst_AdsProcess.bO_StartCappingCanEx
    RoundedRectangle (90,140 20x20), colour toggle: mInst_AdsProcess.bO_StartCappingExec
    Ellipse (30,170 20x20), colour toggle: mInst_AdsProcess.bI_StopCapping
        tap mInst_AdsProcess.bI_StopCapping
    RoundedRectangle (60,170 20x20), colour toggle: mInst_AdsProcess.bO_StopCappingCanEx
    RoundedRectangle (90,170 20x20), colour toggle: mInst_AdsProcess.bO_StopCappingExec
    Ellipse (30,200 20x20), colour toggle: mInst_AdsProcess.bI_Maintenance
        tap mInst_AdsProcess.bI_Maintenance
    RoundedRectangle (60,200 20x20), colour toggle: mInst_AdsProcess.bO_MaintenanceCanEx
    RoundedRectangle (90,200 20x20), colour toggle: mInst_AdsProcess.bO_MaintenanceExec
    Rectangle (130,290 90x20), "Abort"
    Ellipse (30,290 20x20), colour toggle: mInst_AdsProcess.bI_Abort
        tap mInst_AdsProcess.bI_Abort
    RoundedRectangle (60,290 20x20), colour toggle: mInst_AdsProcess.bO_AbortCanEx
    RoundedRectangle (90,290 20x20), colour toggle: mInst_AdsProcess.bO_AbortExec
    RoundedRectangle (90,350 20x20), colour toggle: mInst_AdsProcess.bO_Busy
    Rectangle (120,350 120x20), "Busy"
    Rectangle (20,400 150x20)
    Rectangle (40,400 130x20), "ADS Settings"
    Polyline (40,360)
    RoundedRectangle (340,90 20x20), colour toggle: mInst.bI_Emergency
    Rectangle (370,30 180x20), "not engaged (Service)"
    Rectangle (505,460 80x20), "%1.1f", text variable: mInst_AdsCU.sO_AxisPosition.fO_Val
    Rectangle (505,480 80x20), "%1.1f", text variable: mInst_AdsCH.sO_AxisPosition.fO_Val
    Rectangle (505,500 80x20), "%1.1f", text variable: mInst_AdsPU.sO_AxisPosition.fO_Val
    Ellipse (600,460 20x20), colour toggle: mInst_AdsCU.bO_Ready
    Ellipse (640,460 20x20), colour toggle: mInst_AdsCU.bO_Busy
    Ellipse (600,480 20x20), colour toggle: mInst_AdsCH.bO_Ready
    Ellipse (640,480 20x20), colour toggle: mInst_AdsCH.bO_Busy
    Ellipse (600,500 20x20), colour toggle: mInst_AdsPU.bO_Ready
    Ellipse (640,500 20x20), colour toggle: mInst_AdsPU.bO_Busy
    Rectangle (590,430 40x20), "Ready"
    Rectangle (630,430 40x20), "Busy"
    Rectangle (505,430 83x20), "Position [mm]"
    Rectangle (340,401 150x20)
    Rectangle (360,400 130x20), "ADS Axis Position"
    Ellipse (600,520 20x20), colour toggle: mInst_AdsPurge.bO_Ready
    Ellipse (640,520 20x20), colour toggle: mInst_AdsPurge.bO_Busy
    Rectangle (345,520 150x20), "Purge"
    Ellipse (680,459 20x20), colour toggle: mInst_AdsCU.bO_Error
        toggle mInst_AdsCU.bI_FaultAck
    Ellipse (680,479 20x20), colour toggle: mInst_AdsCH.bO_Error
        toggle mInst_AdsCH.bI_FaultAck
    Ellipse (680,499 20x20), colour toggle: mInst_AdsPU.bO_Error
        tap mInst_AdsPU.bI_FaultAck
    Rectangle (670,430 40x20), "Error"
    Ellipse (680,519 20x20), colour toggle: mInst_AdsPurge.bO_Error
    RoundedRectangle (340,60 20x20), colour toggle: NOT mInst.bI_SafetyOk
    RoundedRectangle (340,30 20x20), colour toggle: mInst.bI_UsrService
    Rectangle (370,60 80x20), "Safety"
    Rectangle (370,90 80x20), "EStop"
    Rectangle (345,460 150x20), "Clean unit (max %d)", text variable: mInst_AdsCU.sO_AxisPosition.fC_Max
    Rectangle (345,480 150x20), "Clean head (max %d)", text variable: mInst_AdsCH.sO_AxisPosition.fC_Max
    Rectangle (345,500 150x20), "Print unit (max %d)", text variable: mInst_AdsPU.sO_AxisPosition.fC_Max
    Rectangle (460,110 100x20), "%d", text variable: mInst.sL_CurrentState^.iL_CurrentStep
    Rectangle (570,110 100x20), "Current step"
    RoundedRectangle (540,140 20x20), colour toggle: mInst.sL_CurrentState^.bL_DevOpActive
    Rectangle (570,140 100x20), "DevOpActive"
    Rectangle (130,430 103x20), "Automatic Mode"
    Ellipse (30,430 20x20), colour toggle: mInst_AdsProcess.bI_AutoMode
        toggle mInst_AdsProcess.bI_AutoMode
    Rectangle (130,460 150x20), "Clean after Capping"
    Ellipse (30,460 20x20), colour toggle: mInst_AdsProcess.bI_CleanAfterCapp
        toggle mInst_AdsProcess.bI_CleanAfterCapp
    Rectangle (130,520 150x20), "Clean after Purge"
    Ellipse (30,520 20x20), colour toggle: mInst_AdsProcess.bI_CleanAfterPurge
        toggle mInst_AdsProcess.bI_CleanAfterPurge
    Rectangle (130,490 150x20), "Purge after Capping"
    Ellipse (30,490 20x20), colour toggle: mInst_AdsProcess.bI_PurgeAfterCapp
        toggle mInst_AdsProcess.bI_PurgeAfterCapp
    Rectangle (130,260 90x20), "Acknowledge"
    Ellipse (30,260 20x20), colour toggle: mInst_AdsProcess.bI_Maintenance
        tap mInst_AdsProcess.bI_AcknowledgeError
    Polyline (480,130), invisible if: NOT _bShutterExist
    Rectangle (431,210 81x20), "Force Open", invisible if: NOT _bShutterExist
    Ellipse (360,210 20x20), invisible if: NOT _bShutterExist
        toggle mInst_FbShutter.bI_ForceInletOpen
    Rectangle (430,240 82x20), "Force Close", invisible if: NOT _bShutterExist
    Ellipse (360,240 20x20), invisible if: NOT _bShutterExist
        toggle mInst_FbShutter.bI_ForceInletClose
    Rectangle (340,170 150x20), invisible if: NOT _bShutterExist
    Rectangle (360,170 130x20), "Shutter", invisible if: NOT _bShutterExist
    RoundedRectangle (530,240 20x20), colour toggle: mInst_FbShutter.bI_ShutterInletClosed, invisible if: NOT _bShutterExist
    Ellipse (390,210 20x20), invisible if: NOT _bShutterExist
        toggle mInst_FbShutter.bI_ForceOutletOpen
    Ellipse (390,240 20x20), invisible if: NOT _bShutterExist
        toggle mInst_FbShutter.bI_ForceOutletClose
    RoundedRectangle (560,240 20x20), colour toggle: mInst_FbShutter.bI_ShutterOutletClosed, invisible if: NOT _bShutterExist
    Rectangle (360,190 81x20), "In Out", invisible if: NOT _bShutterExist
    Rectangle (130,230 90x20), "Open Shutter", invisible if: NOT _bShutterExist
    Ellipse (30,230 20x20), invisible if: NOT _bShutterExist
        tap mInst_AdsProcess.bI_OpenShutter
    RoundedRectangle (60,230 20x20), colour toggle: mInst_AdsProcess.bO_OpenShutterCanEx, invisible if: NOT _bShutterExist
    RoundedRectangle (90,230 20x20), colour toggle: mInst_AdsProcess.bO_OpenShutterExec, invisible if: NOT _bShutterExist
    Ellipse (600,540 20x20), colour toggle: mInst_AdsShutter.bO_Ready, invisible if: NOT _bShutterExist
    Ellipse (640,540 20x20), colour toggle: mInst_AdsShutter.bO_Busy, invisible if: NOT _bShutterExist
    Rectangle (345,540 150x20), "Shutter", invisible if: NOT _bShutterExist
    Ellipse (680,539 20x20), colour toggle: mInst_AdsShutter.bO_Error, invisible if: NOT _bShutterExist
END_VISUALIZATION

